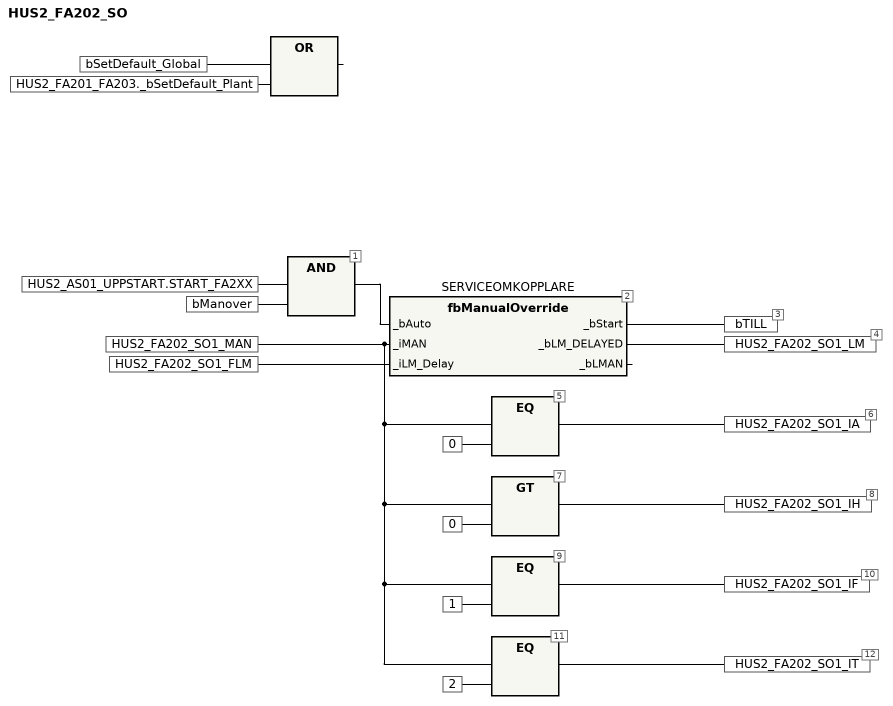
_CFC_ (* Continuous Function Chart, elements in execution order *)
#0 OR(bSetDefault_Global, HUS2_FA201_FA203._bSetDefault_Plant)
#1 AND(HUS2_AS01_UPPSTART.START_FA2XX, bManover)
#2 SERVICEOMKOPPLARE:fbManualOverride(_bAuto: #1, _iMAN: HUS2_FA202_SO1_MAN, _iLM_Delay: HUS2_FA202_SO1_FLM)
#3 bTILL <= #2._bStart
#4 HUS2_FA202_SO1_LM <= #2._bLM_DELAYED
#5 EQ(HUS2_FA202_SO1_MAN, 0)
#6 HUS2_FA202_SO1_IA <= #5
#7 GT(HUS2_FA202_SO1_MAN, 0)
#8 HUS2_FA202_SO1_IH <= #7
#9 EQ(HUS2_FA202_SO1_MAN, 1)
#10 HUS2_FA202_SO1_IF <= #9
#11 EQ(HUS2_FA202_SO1_MAN, 2)
#12 HUS2_FA202_SO1_IT <= #11
_END_CFC_
(* the same logic as Structured Text *)
(* result unused: bSetDefault_Global OR HUS2_FA201_FA203._bSetDefault_Plant *)
SERVICEOMKOPPLARE(_bAuto := HUS2_AS01_UPPSTART.START_FA2XX AND bManover, _iMAN := HUS2_FA202_SO1_MAN, _iLM_Delay := HUS2_FA202_SO1_FLM);
bTILL := SERVICEOMKOPPLARE._bStart;
HUS2_FA202_SO1_LM := SERVICEOMKOPPLARE._bLM_DELAYED;
HUS2_FA202_SO1_IA := HUS2_FA202_SO1_MAN = 0;
HUS2_FA202_SO1_IH := HUS2_FA202_SO1_MAN > 0;
HUS2_FA202_SO1_IF := HUS2_FA202_SO1_MAN = 1;
HUS2_FA202_SO1_IT := HUS2_FA202_SO1_MAN = 2;
END_PROGRAM

(* POU SYSTEM/FA201, FA202, FA203/Fläktstyr/HUS2_FA202_FF01, CFC *)
PROGRAM HUS2_FA202_FF01

VAR
	MANHAND: fbManualOverride;





END_VAR
VAR

END_VAR

VAR_INPUT
	_bAuto							:BOOL;(* enable function block *)
END_VAR

VAR_OUTPUT
	_bMANOVER						:BOOL;
	_bLHAND							:BOOL;
END_VAR
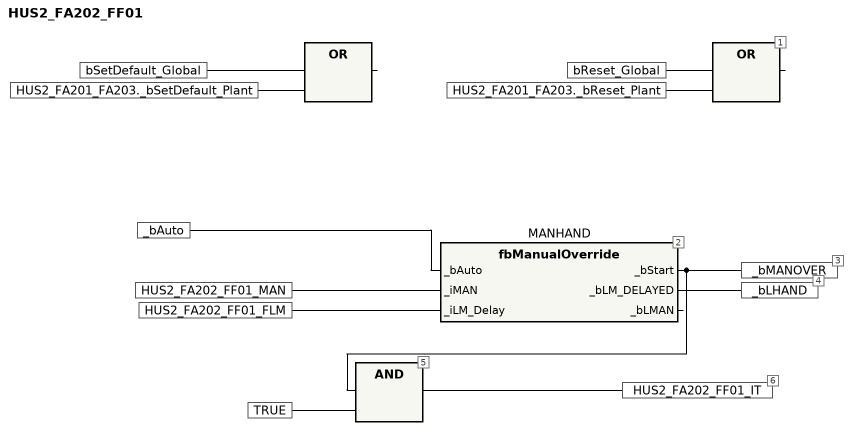
_CFC_ (* Continuous Function Chart, elements in execution order *)
#0 OR(bSetDefault_Global, HUS2_FA201_FA203._bSetDefault_Plant)
#1 OR(bReset_Global, HUS2_FA201_FA203._bReset_Plant)
#2 MANHAND:fbManualOverride(_bAuto: _bAuto, _iMAN: HUS2_FA202_FF01_MAN, _iLM_Delay: HUS2_FA202_FF01_FLM)
#3 _bMANOVER <= #2._bStart
#4 _bLHAND <= #2._bLM_DELAYED
#5 AND(#2._bStart, TRUE)
#6 HUS2_FA202_FF01_IT <= #5
_END_CFC_
(* the same logic as Structured Text *)
(* result unused: bSetDefault_Global OR HUS2_FA201_FA203._bSetDefault_Plant *)
(* result unused: bReset_Global OR HUS2_FA201_FA203._bReset_Plant *)
MANHAND(_bAuto := _bAuto, _iMAN := HUS2_FA202_FF01_MAN, _iLM_Delay := HUS2_FA202_FF01_FLM);
_bMANOVER := MANHAND._bStart;
_bLHAND := MANHAND._bLM_DELAYED;
HUS2_FA202_FF01_IT := MANHAND._bStart AND TRUE;
END_PROGRAM

(* POU SYSTEM/FA201, FA202, FA203/Fläktstyr/HUS2_FA202_FF01_REGLERING, CFC *)
PROGRAM HUS2_FA202_FF01_REGLERING

VAR
	SETRESET: SR;
END_VAR

VAR_INPUT
	bStartFlakt			:BOOL;
	rMV				:REAL;
	rStartForc			:REAL;
	rStoppForc		:REAL;
	rGrundBV			:REAL;
	rForcBV			:REAL;
	bLG				:BOOL;

END_VAR

VAR_OUTPUT
	rSV			:REAL;

END_VAR
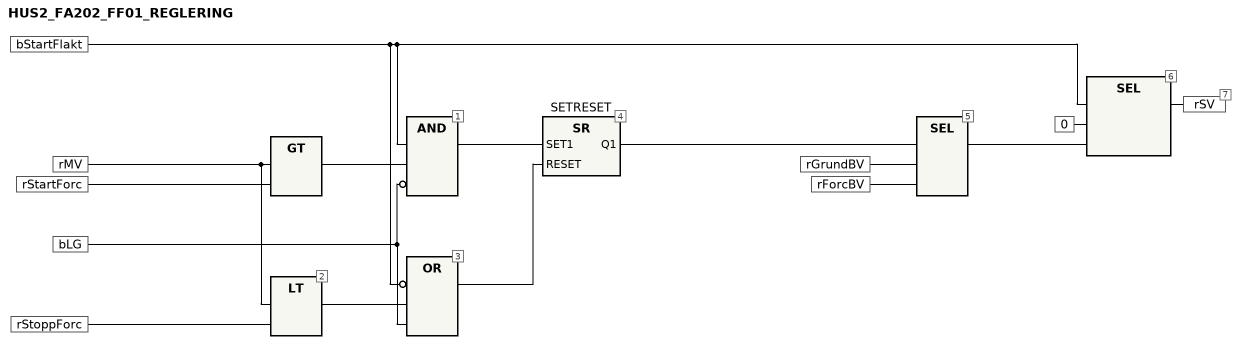
_CFC_ (* Continuous Function Chart, elements in execution order *)
#0 GT(rMV, rStartForc)
#1 AND(bStartFlakt, #0, NOT bLG)
#2 LT(rMV, rStoppForc)
#3 OR(NOT bStartFlakt, #2, bLG)
#4 SETRESET:SR(SET1: #1, RESET: #3)
#5 SEL(#4.Q1, rGrundBV, rForcBV)
#6 SEL(bStartFlakt, 0, #5)
#7 rSV <= #6
_END_CFC_
(* the same logic as Structured Text *)
SETRESET(SET1 := bStartFlakt AND (rMV > rStartForc) AND NOT bLG, RESET := NOT bStartFlakt OR (rMV < rStoppForc) OR bLG);
rSV := SEL(bStartFlakt, 0, SEL(SETRESET.Q1, rGrundBV, rForcBV));
END_PROGRAM

(* POU SYSTEM/FA201, FA202, FA203/Larm/HUS2_FA202_GT51_LARM, FAI *)
PROGRAM HUS2_FA202_GT51_LARM

VAR_OUTPUT
	_bLSumma					: BOOL;	(*Summalarm*)

END_VAR
VAR

	_bSetDefault: 				BOOL;		(*Se default values*)
	fbLarm: fbAvvikelselarm;


	fbHigh: FB_HVACPersistent_Real;
	fbAlarmDelayLH: FB_HVACPersistent_Int;


END_VAR
(* body not read: cfc97 *)
END_PROGRAM

(* POU SYSTEM/FA201, FA202, FA203/HUS2_FA203_SO, CFC *)
PROGRAM HUS2_FA203_SO
VAR_INPUT

	bManover: BOOL;
END_VAR

VAR
	SERVICEOMKOPPLARE: fbManualOverride;

	UPPSTARTSSEKVENSIERING: BOOL;
END_VAR

VAR_OUTPUT
	bTILL:BOOL;

END_VAR
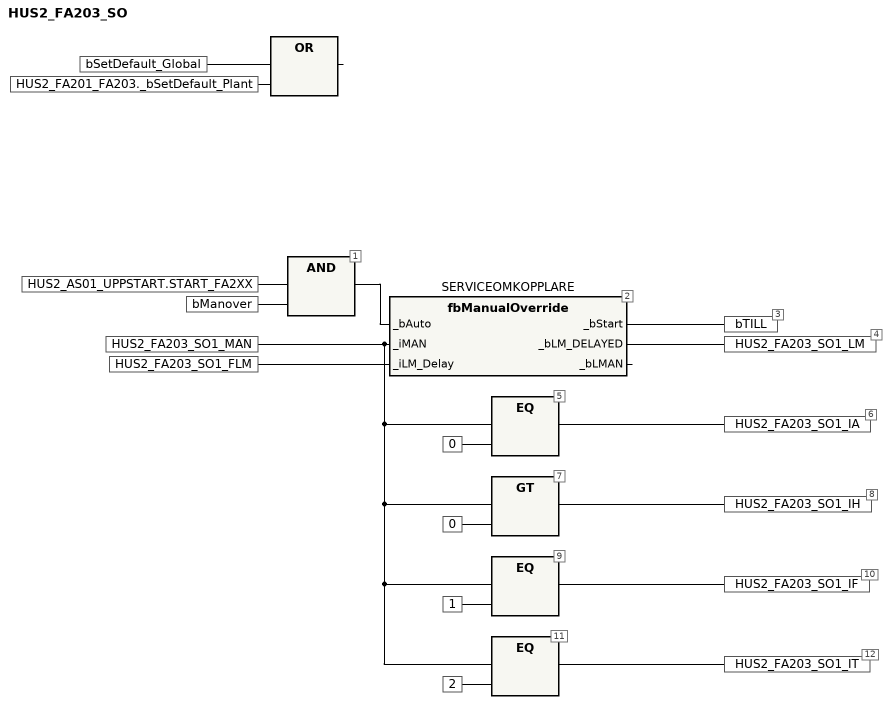
_CFC_ (* Continuous Function Chart, elements in execution order *)
#0 OR(bSetDefault_Global, HUS2_FA201_FA203._bSetDefault_Plant)
#1 AND(HUS2_AS01_UPPSTART.START_FA2XX, bManover)
#2 SERVICEOMKOPPLARE:fbManualOverride(_bAuto: #1, _iMAN: HUS2_FA203_SO1_MAN, _iLM_Delay: HUS2_FA203_SO1_FLM)
#3 bTILL <= #2._bStart
#4 HUS2_FA203_SO1_LM <= #2._bLM_DELAYED
#5 EQ(HUS2_FA203_SO1_MAN, 0)
#6 HUS2_FA203_SO1_IA <= #5
#7 GT(HUS2_FA203_SO1_MAN, 0)
#8 HUS2_FA203_SO1_IH <= #7
#9 EQ(HUS2_FA203_SO1_MAN, 1)
#10 HUS2_FA203_SO1_IF <= #9
#11 EQ(HUS2_FA203_SO1_MAN, 2)
#12 HUS2_FA203_SO1_IT <= #11
_END_CFC_
(* the same logic as Structured Text *)
(* result unused: bSetDefault_Global OR HUS2_FA201_FA203._bSetDefault_Plant *)
SERVICEOMKOPPLARE(_bAuto := HUS2_AS01_UPPSTART.START_FA2XX AND bManover, _iMAN := HUS2_FA203_SO1_MAN, _iLM_Delay := HUS2_FA203_SO1_FLM);
bTILL := SERVICEOMKOPPLARE._bStart;
HUS2_FA203_SO1_LM := SERVICEOMKOPPLARE._bLM_DELAYED;
HUS2_FA203_SO1_IA := HUS2_FA203_SO1_MAN = 0;
HUS2_FA203_SO1_IH := HUS2_FA203_SO1_MAN > 0;
HUS2_FA203_SO1_IF := HUS2_FA203_SO1_MAN = 1;
HUS2_FA203_SO1_IT := HUS2_FA203_SO1_MAN = 2;
END_PROGRAM

(* POU SYSTEM/FA201, FA202, FA203/Fläktstyr/HUS2_FA203_FF01, CFC *)
PROGRAM HUS2_FA203_FF01

VAR
	MANHAND: fbManualOverride;





END_VAR
VAR

END_VAR

VAR_INPUT
	_bAuto							:BOOL;(* enable function block *)
END_VAR

VAR_OUTPUT
	_bMANOVER						:BOOL;
	_bLHAND							:BOOL;
END_VAR
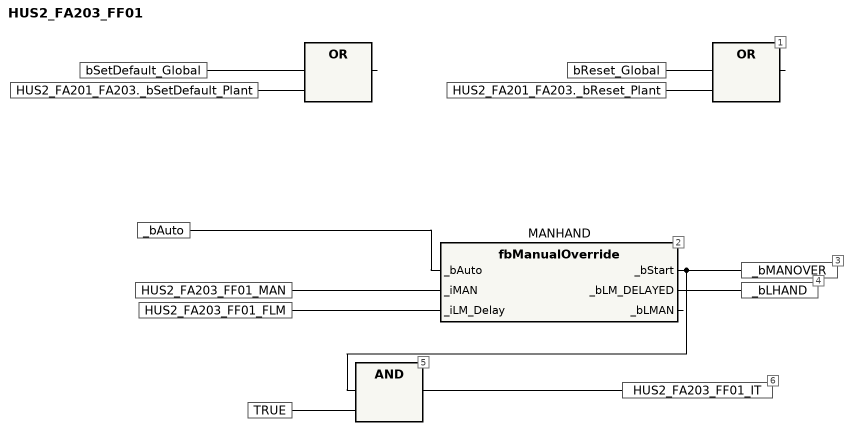
_CFC_ (* Continuous Function Chart, elements in execution order *)
#0 OR(bSetDefault_Global, HUS2_FA201_FA203._bSetDefault_Plant)
#1 OR(bReset_Global, HUS2_FA201_FA203._bReset_Plant)
#2 MANHAND:fbManualOverride(_bAuto: _bAuto, _iMAN: HUS2_FA203_FF01_MAN, _iLM_Delay: HUS2_FA203_FF01_FLM)
#3 _bMANOVER <= #2._bStart
#4 _bLHAND <= #2._bLM_DELAYED
#5 AND(#2._bStart, TRUE)
#6 HUS2_FA203_FF01_IT <= #5
_END_CFC_
(* the same logic as Structured Text *)
(* result unused: bSetDefault_Global OR HUS2_FA201_FA203._bSetDefault_Plant *)
(* result unused: bReset_Global OR HUS2_FA201_FA203._bReset_Plant *)
MANHAND(_bAuto := _bAuto, _iMAN := HUS2_FA203_FF01_MAN, _iLM_Delay := HUS2_FA203_FF01_FLM);
_bMANOVER := MANHAND._bStart;
_bLHAND := MANHAND._bLM_DELAYED;
HUS2_FA203_FF01_IT := MANHAND._bStart AND TRUE;
END_PROGRAM

(* POU SYSTEM/FA201, FA202, FA203/Fläktstyr/HUS2_FA203_FF01_REGLERING, CFC *)
PROGRAM HUS2_FA203_FF01_REGLERING

VAR
	SETRESET: SR;
END_VAR

VAR_INPUT
	bStartFlakt			:BOOL;
	rMV				:REAL;
	rStartForc			:REAL;
	rStoppForc		:REAL;
	rGrundBV			:REAL;
	rForcBV			:REAL;
	bLG				:BOOL;

END_VAR

VAR_OUTPUT
	rSV			:REAL;

END_VAR
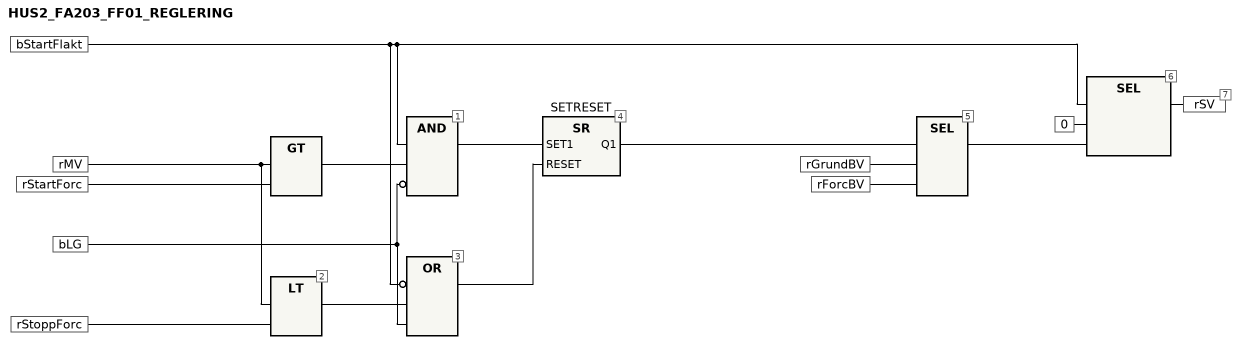
_CFC_ (* Continuous Function Chart, elements in execution order *)
#0 GT(rMV, rStartForc)
#1 AND(bStartFlakt, #0, NOT bLG)
#2 LT(rMV, rStoppForc)
#3 OR(NOT bStartFlakt, #2, bLG)
#4 SETRESET:SR(SET1: #1, RESET: #3)
#5 SEL(#4.Q1, rGrundBV, rForcBV)
#6 SEL(bStartFlakt, 0, #5)
#7 rSV <= #6
_END_CFC_
(* the same logic as Structured Text *)
SETRESET(SET1 := bStartFlakt AND (rMV > rStartForc) AND NOT bLG, RESET := NOT bStartFlakt OR (rMV < rStoppForc) OR bLG);
rSV := SEL(bStartFlakt, 0, SEL(SETRESET.Q1, rGrundBV, rForcBV));
END_PROGRAM

(* POU SYSTEM/FA201, FA202, FA203/Larm/HUS2_FA203_GT51_LARM, FAI *)
PROGRAM HUS2_FA203_GT51_LARM

VAR_OUTPUT
	_bLSumma					: BOOL;	(*Summalarm*)

END_VAR
VAR

	_bSetDefault: 				BOOL;		(*Se default values*)
	fbLarm: fbAvvikelselarm;


	fbHigh: FB_HVACPersistent_Real;
	fbAlarmDelayLH: FB_HVACPersistent_Int;


END_VAR
(* body not read: cfc97 *)
END_PROGRAM

(* POU SYSTEM/FA301, FA302, FA303/HUS3_FA301_FA303, CFC *)
PROGRAM HUS3_FA301_FA303
VAR
	_bSetDefault_Plant		:BOOL;
	_bReset_Plant				:BOOL;

	HUS3_FA301_FF01_M: BOOL;
	HUS3_FA302_FF01_M: BOOL;
	HUS3_FA303_FF01_M: BOOL;
	OVERRIDE_FA301: fbManualOverrideAnalog;
	OVERRIDE_FA302: fbManualOverrideAnalog;
	OVERRIDE_FA303: fbManualOverrideAnalog;
END_VAR
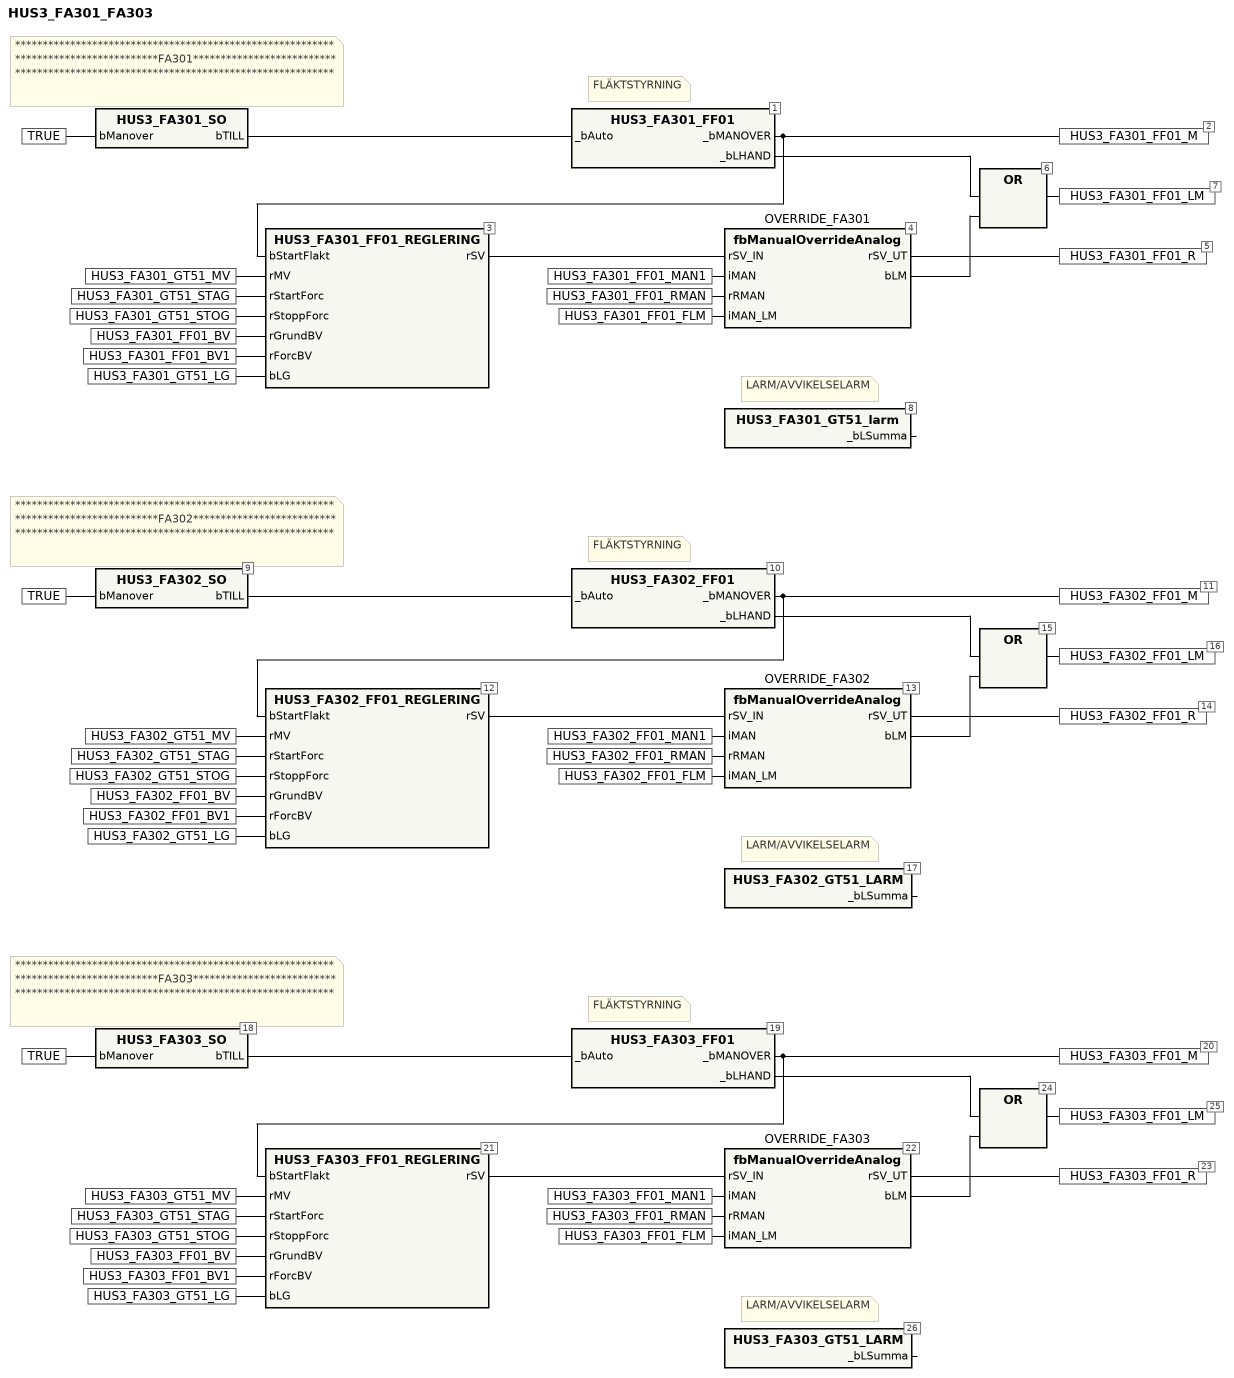
_CFC_ (* Continuous Function Chart, elements in execution order *)
(* LARM/AVVIKELSELARM *)
(* FLÄKTSTYRNING *)
(* ************************************************************************************FA303************************************************************************************ *)
(* LARM/AVVIKELSELARM *)
(* FLÄKTSTYRNING *)
(* LARM/AVVIKELSELARM *)
(* FLÄKTSTYRNING *)
(* ************************************************************************************FA302************************************************************************************ *)
(* ************************************************************************************FA301************************************************************************************ *)
#0 HUS3_FA301_SO(bManover: TRUE)
#1 HUS3_FA301_FF01(_bAuto: #0.bTILL)
#2 HUS3_FA301_FF01_M <= #1._bMANOVER
#3 HUS3_FA301_FF01_REGLERING(bStartFlakt: #1._bMANOVER, rMV: HUS3_FA301_GT51_MV, rStartForc: HUS3_FA301_GT51_STAG, rStoppForc: HUS3_FA301_GT51_STOG, rGrundBV: HUS3_FA301_FF01_BV, rForcBV: HUS3_FA301_FF01_BV1, bLG: HUS3_FA301_GT51_LG)
#4 OVERRIDE_FA301:fbManualOverrideAnalog(rSV_IN: #3.rSV, iMAN: HUS3_FA301_FF01_MAN1, rRMAN: HUS3_FA301_FF01_RMAN, iMAN_LM: HUS3_FA301_FF01_FLM)
#5 HUS3_FA301_FF01_R <= #4.rSV_UT
#6 OR(#1._bLHAND, #4.bLM)
#7 HUS3_FA301_FF01_LM <= #6
#8 HUS3_FA301_GT51_larm()
#9 HUS3_FA302_SO(bManover: TRUE)
#10 HUS3_FA302_FF01(_bAuto: #9.bTILL)
#11 HUS3_FA302_FF01_M <= #10._bMANOVER
#12 HUS3_FA302_FF01_REGLERING(bStartFlakt: #10._bMANOVER, rMV: HUS3_FA302_GT51_MV, rStartForc: HUS3_FA302_GT51_STAG, rStoppForc: HUS3_FA302_GT51_STOG, rGrundBV: HUS3_FA302_FF01_BV, rForcBV: HUS3_FA302_FF01_BV1, bLG: HUS3_FA302_GT51_LG)
#13 OVERRIDE_FA302:fbManualOverrideAnalog(rSV_IN: #12.rSV, iMAN: HUS3_FA302_FF01_MAN1, rRMAN: HUS3_FA302_FF01_RMAN, iMAN_LM: HUS3_FA302_FF01_FLM)
#14 HUS3_FA302_FF01_R <= #13.rSV_UT
#15 OR(#10._bLHAND, #13.bLM)
#16 HUS3_FA302_FF01_LM <= #15
#17 HUS3_FA302_GT51_LARM()
#18 HUS3_FA303_SO(bManover: TRUE)
#19 HUS3_FA303_FF01(_bAuto: #18.bTILL)
#20 HUS3_FA303_FF01_M <= #19._bMANOVER
#21 HUS3_FA303_FF01_REGLERING(bStartFlakt: #19._bMANOVER, rMV: HUS3_FA303_GT51_MV, rStartForc: HUS3_FA303_GT51_STAG, rStoppForc: HUS3_FA303_GT51_STOG, rGrundBV: HUS3_FA303_FF01_BV, rForcBV: HUS3_FA303_FF01_BV1, bLG: HUS3_FA303_GT51_LG)
#22 OVERRIDE_FA303:fbManualOverrideAnalog(rSV_IN: #21.rSV, iMAN: HUS3_FA303_FF01_MAN1, rRMAN: HUS3_FA303_FF01_RMAN, iMAN_LM: HUS3_FA303_FF01_FLM)
#23 HUS3_FA303_FF01_R <= #22.rSV_UT
#24 OR(#19._bLHAND, #22.bLM)
#25 HUS3_FA303_FF01_LM <= #24
#26 HUS3_FA303_GT51_LARM()
_END_CFC_
(* the same logic as Structured Text *)
(* LARM/AVVIKELSELARM *)
(* FLÄKTSTYRNING *)
(* ************************************************************************************FA303************************************************************************************ *)
(* LARM/AVVIKELSELARM *)
(* FLÄKTSTYRNING *)
(* LARM/AVVIKELSELARM *)
(* FLÄKTSTYRNING *)
(* ************************************************************************************FA302************************************************************************************ *)
(* ************************************************************************************FA301************************************************************************************ *)
HUS3_FA301_SO(bManover := TRUE);
HUS3_FA301_FF01(_bAuto := HUS3_FA301_SO.bTILL);
HUS3_FA301_FF01_M := HUS3_FA301_FF01._bMANOVER;
HUS3_FA301_FF01_REGLERING(bStartFlakt := HUS3_FA301_FF01._bMANOVER, rMV := HUS3_FA301_GT51_MV, rStartForc := HUS3_FA301_GT51_STAG, rStoppForc := HUS3_FA301_GT51_STOG, rGrundBV := HUS3_FA301_FF01_BV, rForcBV := HUS3_FA301_FF01_BV1, bLG := HUS3_FA301_GT51_LG);
OVERRIDE_FA301(rSV_IN := HUS3_FA301_FF01_REGLERING.rSV, iMAN := HUS3_FA301_FF01_MAN1, rRMAN := HUS3_FA301_FF01_RMAN, iMAN_LM := HUS3_FA301_FF01_FLM);
HUS3_FA301_FF01_R := OVERRIDE_FA301.rSV_UT;
HUS3_FA301_FF01_LM := HUS3_FA301_FF01._bLHAND OR OVERRIDE_FA301.bLM;
HUS3_FA301_GT51_larm();
HUS3_FA302_SO(bManover := TRUE);
HUS3_FA302_FF01(_bAuto := HUS3_FA302_SO.bTILL);
HUS3_FA302_FF01_M := HUS3_FA302_FF01._bMANOVER;
HUS3_FA302_FF01_REGLERING(bStartFlakt := HUS3_FA302_FF01._bMANOVER, rMV := HUS3_FA302_GT51_MV, rStartForc := HUS3_FA302_GT51_STAG, rStoppForc := HUS3_FA302_GT51_STOG, rGrundBV := HUS3_FA302_FF01_BV, rForcBV := HUS3_FA302_FF01_BV1, bLG := HUS3_FA302_GT51_LG);
OVERRIDE_FA302(rSV_IN := HUS3_FA302_FF01_REGLERING.rSV, iMAN := HUS3_FA302_FF01_MAN1, rRMAN := HUS3_FA302_FF01_RMAN, iMAN_LM := HUS3_FA302_FF01_FLM);
HUS3_FA302_FF01_R := OVERRIDE_FA302.rSV_UT;
HUS3_FA302_FF01_LM := HUS3_FA302_FF01._bLHAND OR OVERRIDE_FA302.bLM;
HUS3_FA302_GT51_LARM();
HUS3_FA303_SO(bManover := TRUE);
HUS3_FA303_FF01(_bAuto := HUS3_FA303_SO.bTILL);
HUS3_FA303_FF01_M := HUS3_FA303_FF01._bMANOVER;
HUS3_FA303_FF01_REGLERING(bStartFlakt := HUS3_FA303_FF01._bMANOVER, rMV := HUS3_FA303_GT51_MV, rStartForc := HUS3_FA303_GT51_STAG, rStoppForc := HUS3_FA303_GT51_STOG, rGrundBV := HUS3_FA303_FF01_BV, rForcBV := HUS3_FA303_FF01_BV1, bLG := HUS3_FA303_GT51_LG);
OVERRIDE_FA303(rSV_IN := HUS3_FA303_FF01_REGLERING.rSV, iMAN := HUS3_FA303_FF01_MAN1, rRMAN := HUS3_FA303_FF01_RMAN, iMAN_LM := HUS3_FA303_FF01_FLM);
HUS3_FA303_FF01_R := OVERRIDE_FA303.rSV_UT;
HUS3_FA303_FF01_LM := HUS3_FA303_FF01._bLHAND OR OVERRIDE_FA303.bLM;
HUS3_FA303_GT51_LARM();
END_PROGRAM

(* POU SYSTEM/FA301, FA302, FA303/HUS3_FA301_SO, CFC *)
PROGRAM HUS3_FA301_SO
VAR_INPUT

	bManover: BOOL;
END_VAR

VAR
	SERVICEOMKOPPLARE: fbManualOverride;

	UPPSTARTSSEKVENSIERING: BOOL;
END_VAR

VAR_OUTPUT
	bTILL:BOOL;

END_VAR
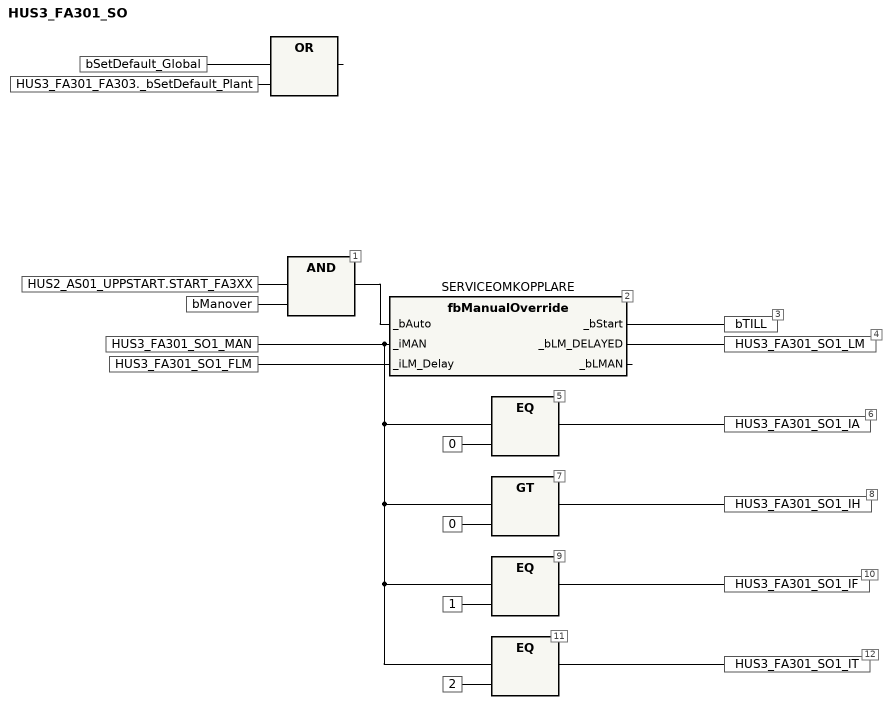
_CFC_ (* Continuous Function Chart, elements in execution order *)
#0 OR(bSetDefault_Global, HUS3_FA301_FA303._bSetDefault_Plant)
#1 AND(HUS2_AS01_UPPSTART.START_FA3XX, bManover)
#2 SERVICEOMKOPPLARE:fbManualOverride(_bAuto: #1, _iMAN: HUS3_FA301_SO1_MAN, _iLM_Delay: HUS3_FA301_SO1_FLM)
#3 bTILL <= #2._bStart
#4 HUS3_FA301_SO1_LM <= #2._bLM_DELAYED
#5 EQ(HUS3_FA301_SO1_MAN, 0)
#6 HUS3_FA301_SO1_IA <= #5
#7 GT(HUS3_FA301_SO1_MAN, 0)
#8 HUS3_FA301_SO1_IH <= #7
#9 EQ(HUS3_FA301_SO1_MAN, 1)
#10 HUS3_FA301_SO1_IF <= #9
#11 EQ(HUS3_FA301_SO1_MAN, 2)
#12 HUS3_FA301_SO1_IT <= #11
_END_CFC_
(* the same logic as Structured Text *)
(* result unused: bSetDefault_Global OR HUS3_FA301_FA303._bSetDefault_Plant *)
SERVICEOMKOPPLARE(_bAuto := HUS2_AS01_UPPSTART.START_FA3XX AND bManover, _iMAN := HUS3_FA301_SO1_MAN, _iLM_Delay := HUS3_FA301_SO1_FLM);
bTILL := SERVICEOMKOPPLARE._bStart;
HUS3_FA301_SO1_LM := SERVICEOMKOPPLARE._bLM_DELAYED;
HUS3_FA301_SO1_IA := HUS3_FA301_SO1_MAN = 0;
HUS3_FA301_SO1_IH := HUS3_FA301_SO1_MAN > 0;
HUS3_FA301_SO1_IF := HUS3_FA301_SO1_MAN = 1;
HUS3_FA301_SO1_IT := HUS3_FA301_SO1_MAN = 2;
END_PROGRAM

(* POU SYSTEM/FA301, FA302, FA303/Fläktstyr/HUS3_FA301_FF01, CFC *)
PROGRAM HUS3_FA301_FF01

VAR
	MANHAND: fbManualOverride;





END_VAR
VAR

END_VAR

VAR_INPUT
	_bAuto							:BOOL;(* enable function block *)
END_VAR

VAR_OUTPUT
	_bMANOVER						:BOOL;
	_bLHAND							:BOOL;
END_VAR
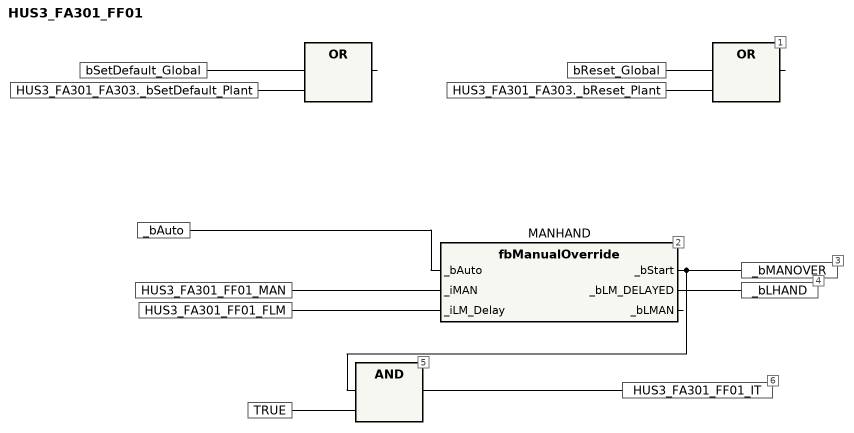
_CFC_ (* Continuous Function Chart, elements in execution order *)
#0 OR(bSetDefault_Global, HUS3_FA301_FA303._bSetDefault_Plant)
#1 OR(bReset_Global, HUS3_FA301_FA303._bReset_Plant)
#2 MANHAND:fbManualOverride(_bAuto: _bAuto, _iMAN: HUS3_FA301_FF01_MAN, _iLM_Delay: HUS3_FA301_FF01_FLM)
#3 _bMANOVER <= #2._bStart
#4 _bLHAND <= #2._bLM_DELAYED
#5 AND(#2._bStart, TRUE)
#6 HUS3_FA301_FF01_IT <= #5
_END_CFC_
(* the same logic as Structured Text *)
(* result unused: bSetDefault_Global OR HUS3_FA301_FA303._bSetDefault_Plant *)
(* result unused: bReset_Global OR HUS3_FA301_FA303._bReset_Plant *)
MANHAND(_bAuto := _bAuto, _iMAN := HUS3_FA301_FF01_MAN, _iLM_Delay := HUS3_FA301_FF01_FLM);
_bMANOVER := MANHAND._bStart;
_bLHAND := MANHAND._bLM_DELAYED;
HUS3_FA301_FF01_IT := MANHAND._bStart AND TRUE;
END_PROGRAM

(* POU SYSTEM/FA301, FA302, FA303/Fläktstyr/HUS3_FA301_FF01_REGLERING, CFC *)
PROGRAM HUS3_FA301_FF01_REGLERING

VAR
	SETRESET: SR;
END_VAR

VAR_INPUT
	bStartFlakt			:BOOL;
	rMV				:REAL;
	rStartForc			:REAL;
	rStoppForc		:REAL;
	rGrundBV			:REAL;
	rForcBV			:REAL;
	bLG				:BOOL;

END_VAR

VAR_OUTPUT
	rSV			:REAL;

END_VAR
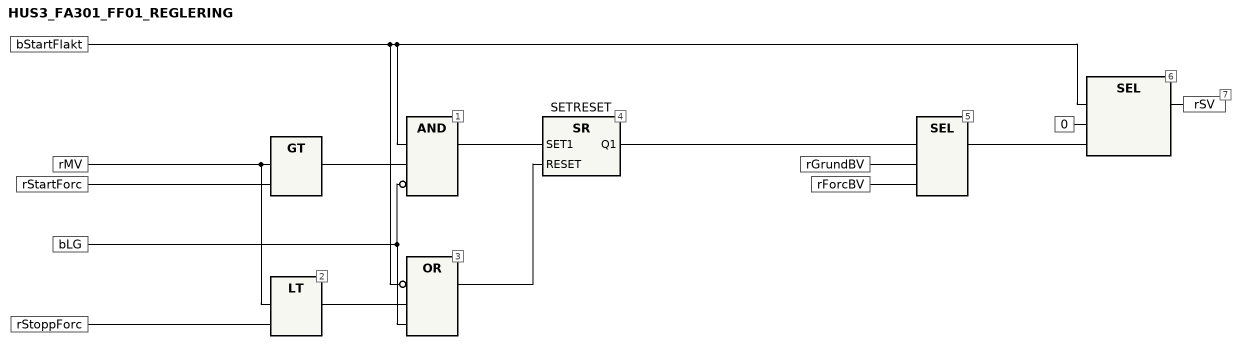
_CFC_ (* Continuous Function Chart, elements in execution order *)
#0 GT(rMV, rStartForc)
#1 AND(bStartFlakt, #0, NOT bLG)
#2 LT(rMV, rStoppForc)
#3 OR(NOT bStartFlakt, #2, bLG)
#4 SETRESET:SR(SET1: #1, RESET: #3)
#5 SEL(#4.Q1, rGrundBV, rForcBV)
#6 SEL(bStartFlakt, 0, #5)
#7 rSV <= #6
_END_CFC_
(* the same logic as Structured Text *)
SETRESET(SET1 := bStartFlakt AND (rMV > rStartForc) AND NOT bLG, RESET := NOT bStartFlakt OR (rMV < rStoppForc) OR bLG);
rSV := SEL(bStartFlakt, 0, SEL(SETRESET.Q1, rGrundBV, rForcBV));
END_PROGRAM

(* POU SYSTEM/FA301, FA302, FA303/Larm/HUS3_FA301_GT51_LARM, FAI *)
PROGRAM HUS3_FA301_GT51_LARM

VAR_OUTPUT
	_bLSumma					: BOOL;	(*Summalarm*)

END_VAR
VAR

	_bSetDefault: 				BOOL;		(*Se default values*)
	fbLarm: fbAvvikelselarm;


	fbHigh: FB_HVACPersistent_Real;
	fbAlarmDelayLH: FB_HVACPersistent_Int;


END_VAR
(* body not read: cfc97 *)
END_PROGRAM

(* POU SYSTEM/FA301, FA302, FA303/HUS3_FA302_SO, CFC *)
PROGRAM HUS3_FA302_SO
VAR_INPUT

	bManover: BOOL;
END_VAR

VAR
	SERVICEOMKOPPLARE: fbManualOverride;

	UPPSTARTSSEKVENSIERING: BOOL;
END_VAR

VAR_OUTPUT
	bTILL:BOOL;

END_VAR
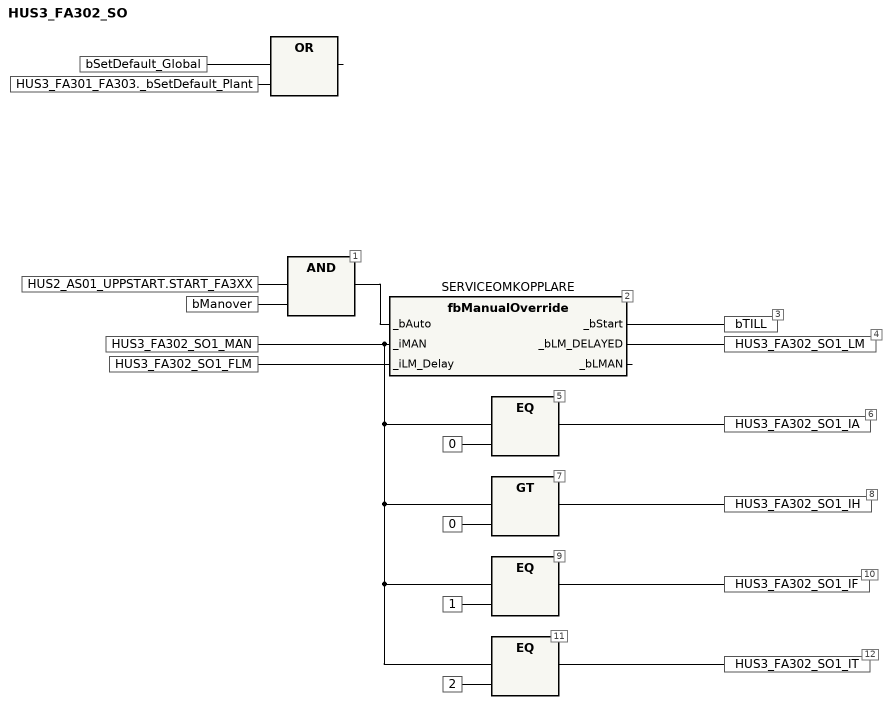
_CFC_ (* Continuous Function Chart, elements in execution order *)
#0 OR(bSetDefault_Global, HUS3_FA301_FA303._bSetDefault_Plant)
#1 AND(HUS2_AS01_UPPSTART.START_FA3XX, bManover)
#2 SERVICEOMKOPPLARE:fbManualOverride(_bAuto: #1, _iMAN: HUS3_FA302_SO1_MAN, _iLM_Delay: HUS3_FA302_SO1_FLM)
#3 bTILL <= #2._bStart
#4 HUS3_FA302_SO1_LM <= #2._bLM_DELAYED
#5 EQ(HUS3_FA302_SO1_MAN, 0)
#6 HUS3_FA302_SO1_IA <= #5
#7 GT(HUS3_FA302_SO1_MAN, 0)
#8 HUS3_FA302_SO1_IH <= #7
#9 EQ(HUS3_FA302_SO1_MAN, 1)
#10 HUS3_FA302_SO1_IF <= #9
#11 EQ(HUS3_FA302_SO1_MAN, 2)
#12 HUS3_FA302_SO1_IT <= #11
_END_CFC_
(* the same logic as Structured Text *)
(* result unused: bSetDefault_Global OR HUS3_FA301_FA303._bSetDefault_Plant *)
SERVICEOMKOPPLARE(_bAuto := HUS2_AS01_UPPSTART.START_FA3XX AND bManover, _iMAN := HUS3_FA302_SO1_MAN, _iLM_Delay := HUS3_FA302_SO1_FLM);
bTILL := SERVICEOMKOPPLARE._bStart;
HUS3_FA302_SO1_LM := SERVICEOMKOPPLARE._bLM_DELAYED;
HUS3_FA302_SO1_IA := HUS3_FA302_SO1_MAN = 0;
HUS3_FA302_SO1_IH := HUS3_FA302_SO1_MAN > 0;
HUS3_FA302_SO1_IF := HUS3_FA302_SO1_MAN = 1;
HUS3_FA302_SO1_IT := HUS3_FA302_SO1_MAN = 2;
END_PROGRAM

(* POU SYSTEM/FA301, FA302, FA303/Fläktstyr/HUS3_FA302_FF01, CFC *)
PROGRAM HUS3_FA302_FF01

VAR
	MANHAND: fbManualOverride;





END_VAR
VAR

END_VAR

VAR_INPUT
	_bAuto							:BOOL;(* enable function block *)
END_VAR

VAR_OUTPUT
	_bMANOVER						:BOOL;
	_bLHAND							:BOOL;
END_VAR
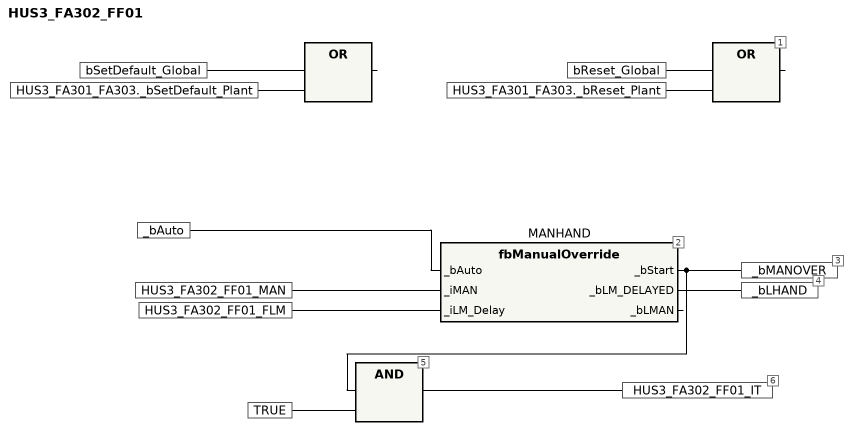
_CFC_ (* Continuous Function Chart, elements in execution order *)
#0 OR(bSetDefault_Global, HUS3_FA301_FA303._bSetDefault_Plant)
#1 OR(bReset_Global, HUS3_FA301_FA303._bReset_Plant)
#2 MANHAND:fbManualOverride(_bAuto: _bAuto, _iMAN: HUS3_FA302_FF01_MAN, _iLM_Delay: HUS3_FA302_FF01_FLM)
#3 _bMANOVER <= #2._bStart
#4 _bLHAND <= #2._bLM_DELAYED
#5 AND(#2._bStart, TRUE)
#6 HUS3_FA302_FF01_IT <= #5
_END_CFC_
(* the same logic as Structured Text *)
(* result unused: bSetDefault_Global OR HUS3_FA301_FA303._bSetDefault_Plant *)
(* result unused: bReset_Global OR HUS3_FA301_FA303._bReset_Plant *)
MANHAND(_bAuto := _bAuto, _iMAN := HUS3_FA302_FF01_MAN, _iLM_Delay := HUS3_FA302_FF01_FLM);
_bMANOVER := MANHAND._bStart;
_bLHAND := MANHAND._bLM_DELAYED;
HUS3_FA302_FF01_IT := MANHAND._bStart AND TRUE;
END_PROGRAM

(* POU SYSTEM/FA301, FA302, FA303/Fläktstyr/HUS3_FA302_FF01_REGLERING, CFC *)
PROGRAM HUS3_FA302_FF01_REGLERING

VAR
	SETRESET: SR;
END_VAR

VAR_INPUT
	bStartFlakt			:BOOL;
	rMV				:REAL;
	rStartForc			:REAL;
	rStoppForc		:REAL;
	rGrundBV			:REAL;
	rForcBV			:REAL;
	bLG				:BOOL;

END_VAR

VAR_OUTPUT
	rSV			:REAL;

END_VAR
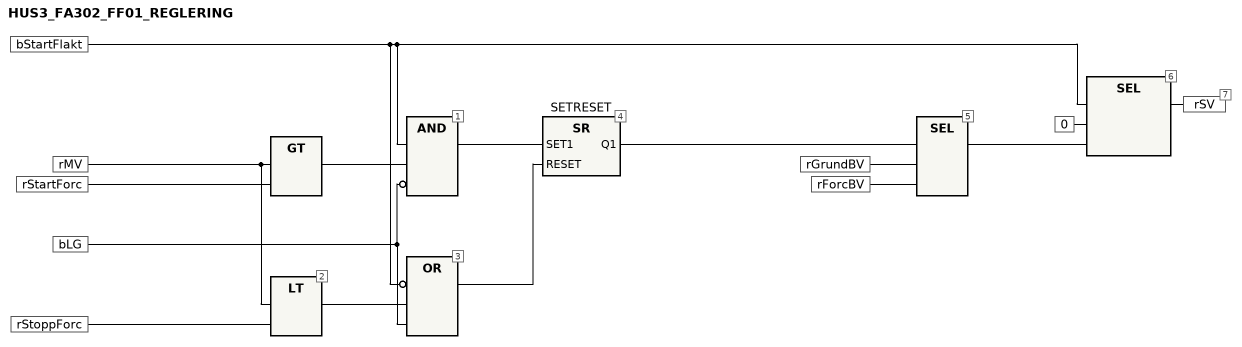
_CFC_ (* Continuous Function Chart, elements in execution order *)
#0 GT(rMV, rStartForc)
#1 AND(bStartFlakt, #0, NOT bLG)
#2 LT(rMV, rStoppForc)
#3 OR(NOT bStartFlakt, #2, bLG)
#4 SETRESET:SR(SET1: #1, RESET: #3)
#5 SEL(#4.Q1, rGrundBV, rForcBV)
#6 SEL(bStartFlakt, 0, #5)
#7 rSV <= #6
_END_CFC_
(* the same logic as Structured Text *)
SETRESET(SET1 := bStartFlakt AND (rMV > rStartForc) AND NOT bLG, RESET := NOT bStartFlakt OR (rMV < rStoppForc) OR bLG);
rSV := SEL(bStartFlakt, 0, SEL(SETRESET.Q1, rGrundBV, rForcBV));
END_PROGRAM

(* POU SYSTEM/FA301, FA302, FA303/Larm/HUS3_FA302_GT51_LARM, FAI *)
PROGRAM HUS3_FA302_GT51_LARM

VAR_OUTPUT
	_bLSumma					: BOOL;	(*Summalarm*)

END_VAR
VAR

	_bSetDefault: 				BOOL;		(*Se default values*)
	fbLarm: fbAvvikelselarm;


	fbHigh: FB_HVACPersistent_Real;
	fbAlarmDelayLH: FB_HVACPersistent_Int;


END_VAR
(* body not read: cfc97 *)
END_PROGRAM

(* POU SYSTEM/FA301, FA302, FA303/HUS3_FA303_SO, CFC *)
PROGRAM HUS3_FA303_SO
VAR_INPUT

	bManover: BOOL;
END_VAR

VAR
	SERVICEOMKOPPLARE: fbManualOverride;

	UPPSTARTSSEKVENSIERING: BOOL;
END_VAR

VAR_OUTPUT
	bTILL:BOOL;

END_VAR
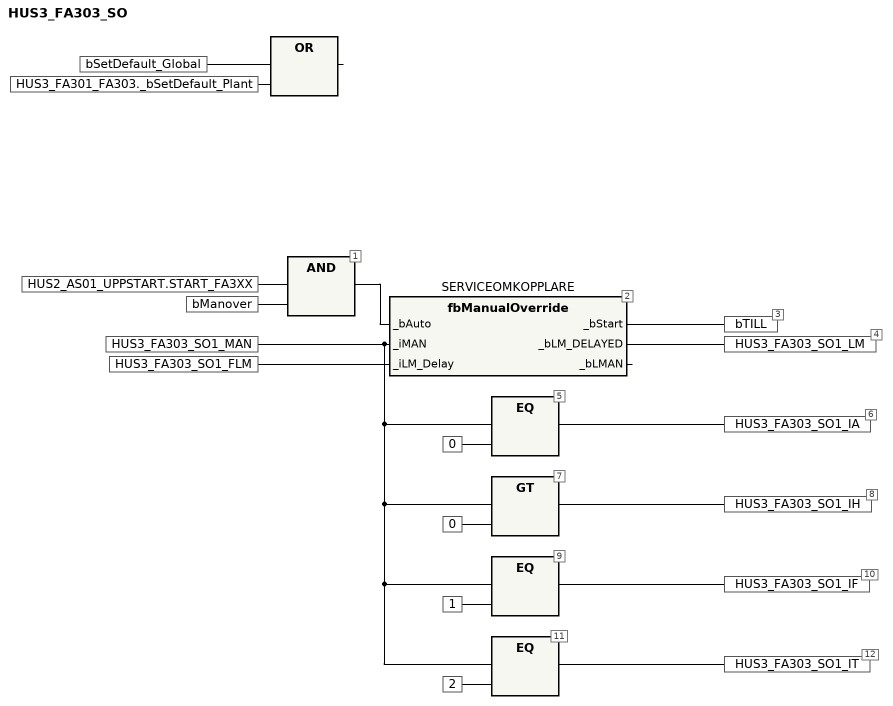
_CFC_ (* Continuous Function Chart, elements in execution order *)
#0 OR(bSetDefault_Global, HUS3_FA301_FA303._bSetDefault_Plant)
#1 AND(HUS2_AS01_UPPSTART.START_FA3XX, bManover)
#2 SERVICEOMKOPPLARE:fbManualOverride(_bAuto: #1, _iMAN: HUS3_FA303_SO1_MAN, _iLM_Delay: HUS3_FA303_SO1_FLM)
#3 bTILL <= #2._bStart
#4 HUS3_FA303_SO1_LM <= #2._bLM_DELAYED
#5 EQ(HUS3_FA303_SO1_MAN, 0)
#6 HUS3_FA303_SO1_IA <= #5
#7 GT(HUS3_FA303_SO1_MAN, 0)
#8 HUS3_FA303_SO1_IH <= #7
#9 EQ(HUS3_FA303_SO1_MAN, 1)
#10 HUS3_FA303_SO1_IF <= #9
#11 EQ(HUS3_FA303_SO1_MAN, 2)
#12 HUS3_FA303_SO1_IT <= #11
_END_CFC_
(* the same logic as Structured Text *)
(* result unused: bSetDefault_Global OR HUS3_FA301_FA303._bSetDefault_Plant *)
SERVICEOMKOPPLARE(_bAuto := HUS2_AS01_UPPSTART.START_FA3XX AND bManover, _iMAN := HUS3_FA303_SO1_MAN, _iLM_Delay := HUS3_FA303_SO1_FLM);
bTILL := SERVICEOMKOPPLARE._bStart;
HUS3_FA303_SO1_LM := SERVICEOMKOPPLARE._bLM_DELAYED;
HUS3_FA303_SO1_IA := HUS3_FA303_SO1_MAN = 0;
HUS3_FA303_SO1_IH := HUS3_FA303_SO1_MAN > 0;
HUS3_FA303_SO1_IF := HUS3_FA303_SO1_MAN = 1;
HUS3_FA303_SO1_IT := HUS3_FA303_SO1_MAN = 2;
END_PROGRAM

(* POU SYSTEM/FA301, FA302, FA303/Fläktstyr/HUS3_FA303_FF01, CFC *)
PROGRAM HUS3_FA303_FF01

VAR
	MANHAND: fbManualOverride;





END_VAR
VAR

END_VAR

VAR_INPUT
	_bAuto							:BOOL;(* enable function block *)
END_VAR

VAR_OUTPUT
	_bMANOVER						:BOOL;
	_bLHAND							:BOOL;
END_VAR
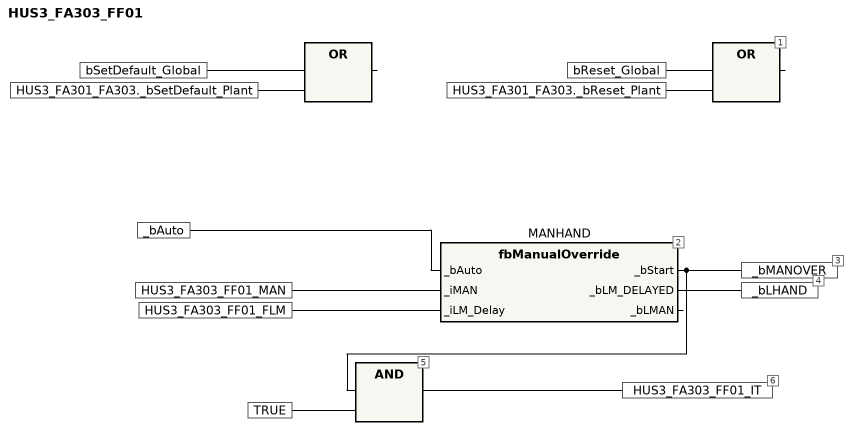
_CFC_ (* Continuous Function Chart, elements in execution order *)
#0 OR(bSetDefault_Global, HUS3_FA301_FA303._bSetDefault_Plant)
#1 OR(bReset_Global, HUS3_FA301_FA303._bReset_Plant)
#2 MANHAND:fbManualOverride(_bAuto: _bAuto, _iMAN: HUS3_FA303_FF01_MAN, _iLM_Delay: HUS3_FA303_FF01_FLM)
#3 _bMANOVER <= #2._bStart
#4 _bLHAND <= #2._bLM_DELAYED
#5 AND(#2._bStart, TRUE)
#6 HUS3_FA303_FF01_IT <= #5
_END_CFC_
(* the same logic as Structured Text *)
(* result unused: bSetDefault_Global OR HUS3_FA301_FA303._bSetDefault_Plant *)
(* result unused: bReset_Global OR HUS3_FA301_FA303._bReset_Plant *)
MANHAND(_bAuto := _bAuto, _iMAN := HUS3_FA303_FF01_MAN, _iLM_Delay := HUS3_FA303_FF01_FLM);
_bMANOVER := MANHAND._bStart;
_bLHAND := MANHAND._bLM_DELAYED;
HUS3_FA303_FF01_IT := MANHAND._bStart AND TRUE;
END_PROGRAM

(* POU SYSTEM/FA301, FA302, FA303/Fläktstyr/HUS3_FA303_FF01_REGLERING, CFC *)
PROGRAM HUS3_FA303_FF01_REGLERING

VAR
	SETRESET: SR;
END_VAR

VAR_INPUT
	bStartFlakt			:BOOL;
	rMV				:REAL;
	rStartForc			:REAL;
	rStoppForc		:REAL;
	rGrundBV			:REAL;
	rForcBV			:REAL;
	bLG				:BOOL;

END_VAR

VAR_OUTPUT
	rSV			:REAL;

END_VAR
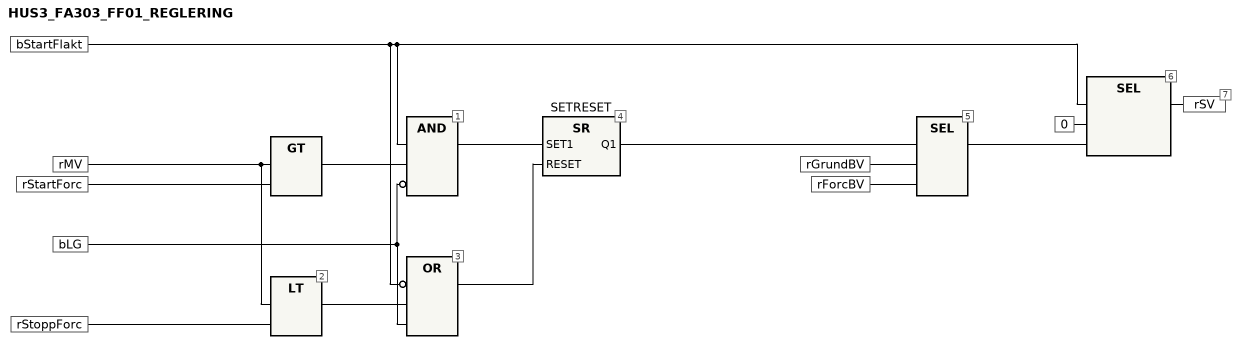
_CFC_ (* Continuous Function Chart, elements in execution order *)
#0 GT(rMV, rStartForc)
#1 AND(bStartFlakt, #0, NOT bLG)
#2 LT(rMV, rStoppForc)
#3 OR(NOT bStartFlakt, #2, bLG)
#4 SETRESET:SR(SET1: #1, RESET: #3)
#5 SEL(#4.Q1, rGrundBV, rForcBV)
#6 SEL(bStartFlakt, 0, #5)
#7 rSV <= #6
_END_CFC_
(* the same logic as Structured Text *)
SETRESET(SET1 := bStartFlakt AND (rMV > rStartForc) AND NOT bLG, RESET := NOT bStartFlakt OR (rMV < rStoppForc) OR bLG);
rSV := SEL(bStartFlakt, 0, SEL(SETRESET.Q1, rGrundBV, rForcBV));
END_PROGRAM

(* POU SYSTEM/FA301, FA302, FA303/Larm/HUS3_FA303_GT51_LARM, FAI *)
PROGRAM HUS3_FA303_GT51_LARM

VAR_OUTPUT
	_bLSumma					: BOOL;	(*Summalarm*)

END_VAR
VAR

	_bSetDefault: 				BOOL;		(*Se default values*)
	fbLarm: fbAvvikelselarm;


	fbHigh: FB_HVACPersistent_Real;
	fbAlarmDelayLH: FB_HVACPersistent_Int;


END_VAR
(* body not read: cfc97 *)
END_PROGRAM

(* POU ReadMe, ST *)
PROGRAM ReadMe
VAR
END_VAR
(*


Oskar Lindström, Automationsbolaget Sverige AB
2020-03-04


*)
END_PROGRAM

(* POU xEgna Funktionsblock/Modbus/Modbusfunktioner_med_Master/_ModbusTCP_Controller, ST *)
FUNCTION_BLOCK _ModbusTCP_Controller

VAR
	stController			: ST_TCP_CONTROLLER:=(iWorkingUnitId:=1);
	pController			: POINTER TO ST_TCP_CONTROLLER;

END_VAR
(* DO NOT CHANGE ANYTHING IN THIS CODE *)

(* Output the pointer to this controller*)
pController := ADR(stController);

(* Do any units exist? *)
IF stController.iNoUnits>0 THEN
	(* Is the current unit done? *)
	IF stController.bUnitIsDone  THEN
		(* Yes, reset the done flag and increase the unit ID counter *)
		stController.bUnitIsDone:=FALSE;
		stController.iWorkingUnitId:=stController.iWorkingUnitId+1;
		(*Handle rollover of the unit ID counter *)
		IF stController.iWorkingUnitId>stController.iNoUnits THEN
			stController.iWorkingUnitId:=1;
		END_IF
	END_IF
END_IF
END_FUNCTION_BLOCK

(* POU xEgna Funktionsblock/Time_to_SCADA/FB_CitectTimeTo_HVAC_1_DATE, ST *)
(*
Funktionsblock för att hantera en tid från Citect/Webport till Beckhoffs tidkanaler
Av: Beckhoff Automation AB Roger Grönvall
Lib: TCHVAC.LIB
*)
FUNCTION_BLOCK FB_CitectTimeTo_HVAC_1_DATE

VAR_INPUT
END_VAR

VAR_IN_OUT
	_iCitect_OnTime:		INT;		(*Time On from HMI*)
	_iCitect_OffTime:		INT;		(*Time Off from HMI*)
END_VAR
VAR_OUTPUT
	_uiOnTime_hh:		UINT;	(*Hours for on time*)
	_uiOnTime_mm:		UINT;	(*Minutes for on time*)
	_uiOffTime_hh:		UINT;	(*Hours for off time*)
	_uiOffTime_mm:		UINT;	(*Minutes for off time*)
	_bEnableTimeCh:		BOOL;	(*Enable timechannel*)
END_VAR
VAR
	iNowOn:				INT;		(*Temp var for on time*)
	iNowOff:				INT;		(*Temp var for off time*)
	fbSaveOnTime:		FB_HVACPersistent_Int;
	fbSaveOffTime:		FB_HVACPersistent_Int;
END_VAR

(*
	This FB converts hmi time from Citect to HVAC TimeChannel
	the input time is an integer. i.e Time 15:46 = _iCitect_OnTime 1546. Then
	the our and minute is extracted to the HVAC time. 
	No erreor handling if time is not in the appropriate range.
	Maybe the persistent data handling for the TC needs to be disabled
*)
(*Get the on time*)
iNowOn := _iCitect_OnTime;
(*Get hour*)
_uiOnTime_hh := iNowOn / 100;
(*Get minute*)
_uiOnTime_mm := iNowOn - ( _uiOnTime_hh * 100);


(*Get the off time*)
iNowOff := _iCitect_OffTime;
(*Get hour*)
_uiOffTime_hh := iNowOff / 100;
(*Get minute*)
_uiOffTime_mm := iNowOff - ( _uiOffTime_hh * 100);


(*Find out if we have some time set, then enable the output*)
IF  _iCitect_OnTime > 0 THEN
	_bEnableTimeCh := TRUE;
ELSE
	_bEnableTimeCh := FALSE;
END_IF


(*Save the on/off time data persistent*)
fbSaveOnTime(bSetDefault:= , iVar_Default:= , iVar:= _iCitect_OnTime );
fbSaveOffTime(bSetDefault:= , iVar_Default:= , iVar:= _iCitect_OffTime );
END_FUNCTION_BLOCK

(* POU xEgna Funktionsblock/fbActiveLG, CFC *)
FUNCTION_BLOCK fbActiveLG
VAR_INPUT
	rMV:REAL;
	rHighLimit:REAL;
	rLowLimit:REAL;
	iLG_FL:INT;
END_VAR
VAR_OUTPUT
	bLG:BOOL;
END_VAR
VAR
	FBTON1: TON;
END_VAR
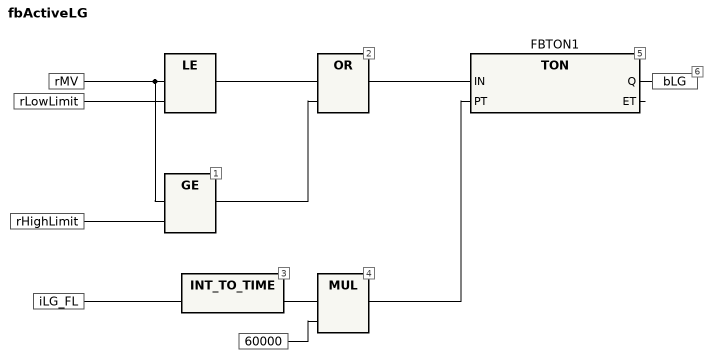
_CFC_ (* Continuous Function Chart, elements in execution order *)
#0 LE(rMV, rLowLimit)
#1 GE(rMV, rHighLimit)
#2 OR(#0, #1)
#3 INT_TO_TIME(iLG_FL)
#4 MUL(#3, 60000)
#5 FBTON1:TON(IN: #2, PT: #4)
#6 bLG <= #5.Q
_END_CFC_
(* the same logic as Structured Text *)
FBTON1(IN := (rMV <= rLowLimit) OR (rMV >= rHighLimit), PT := INT_TO_TIME(iLG_FL) * 60000);
bLG := FBTON1.Q;
END_FUNCTION_BLOCK

(* POU xEgna Funktionsblock/fbAvvikelselarm_SEC, CFC *)
FUNCTION_BLOCK fbAvvikelselarm_SEC
VAR
	TON1: TON;
	TON2: TON;
END_VAR
VAR_INPUT
	_rBB: REAL;
	_rMV: REAL;
	_rLL: REAL;
	_iFLL: INT;
	_rLH: REAL;
	_iFLH: INT;
	_bAktiveraLarm: BOOL;

END_VAR


VAR_OUTPUT
	_bLL: BOOL;
	_bLH: BOOL;
	_bLSummA: BOOL;
END_VAR
VAR (* helpers for the ST form of the networks *)
	_t54 : TIME;
END_VAR
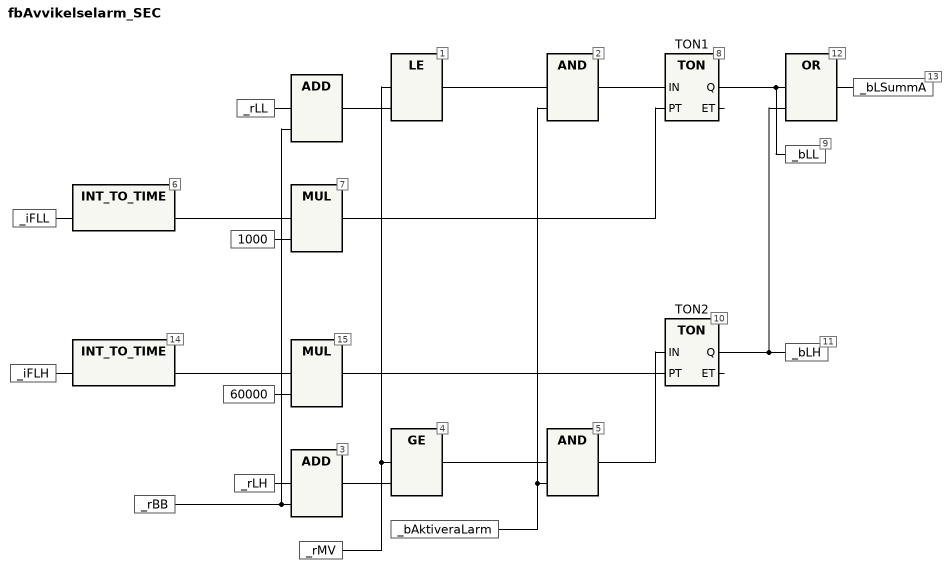
_CFC_ (* Continuous Function Chart, elements in execution order *)
#0 ADD(_rLL, _rBB)
#1 LE(_rMV, #0)
#2 AND(#1, _bAktiveraLarm)
#3 ADD(_rLH, _rBB)
#4 GE(_rMV, #3)
#5 AND(#4, _bAktiveraLarm)
#6 INT_TO_TIME(_iFLL)
#7 MUL(#6, 1000)
#8 TON1:TON(IN: #2, PT: #7)
#9 _bLL <= #8.Q
#10 TON2:TON(IN: #5, PT: #15)
#11 _bLH <= #10.Q
#12 OR(#8.Q, #10.Q)
#13 _bLSummA <= #12
#14 INT_TO_TIME(_iFLH)
#15 MUL(#14, 60000)
_END_CFC_
(* the same logic as Structured Text *)
TON1(IN := (_rMV <= (_rLL + _rBB)) AND _bAktiveraLarm, PT := INT_TO_TIME(_iFLL) * 1000);
_bLL := TON1.Q;
TON2(IN := (_rMV >= (_rLH + _rBB)) AND _bAktiveraLarm, PT := _t54);
_bLH := TON2.Q;
_bLSummA := TON1.Q OR TON2.Q;
_t54 := INT_TO_TIME(_iFLH) * 60000;
END_FUNCTION_BLOCK

(* POU xEgna Funktionsblock/fbAvvikelselarmLA, CFC *)
FUNCTION_BLOCK fbAvvikelselarmLA
VAR
	TON1: TON;
	TON2: TON;
END_VAR
VAR_INPUT
	_rBB: REAL;
	_rMV: REAL;
	_rLA: REAL;
	_iFLA: INT;
	_bAktiveraLarm: BOOL;

END_VAR


VAR_OUTPUT
	_bLA: BOOL;
END_VAR
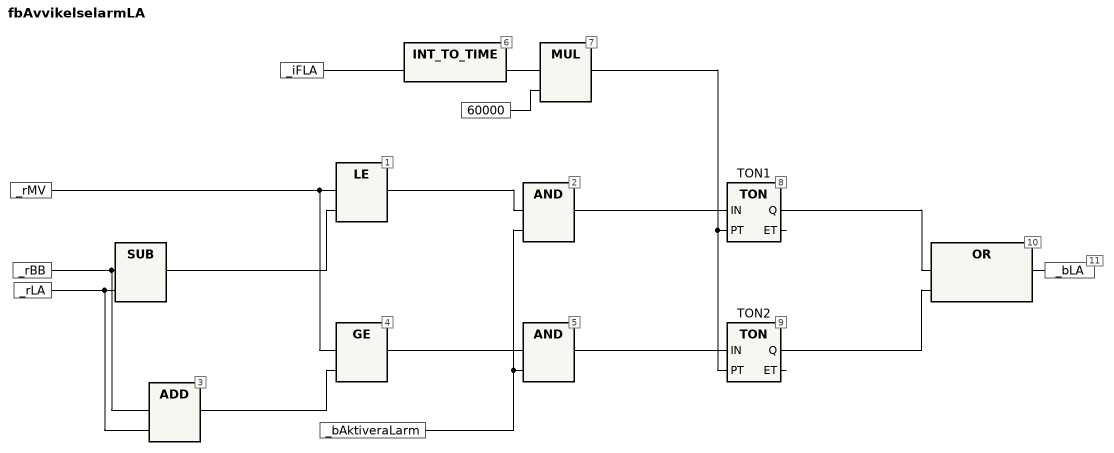
_CFC_ (* Continuous Function Chart, elements in execution order *)
#0 SUB(_rBB, _rLA)
#1 LE(_rMV, #0)
#2 AND(#1, _bAktiveraLarm)
#3 ADD(_rBB, _rLA)
#4 GE(_rMV, #3)
#5 AND(#4, _bAktiveraLarm)
#6 INT_TO_TIME(_iFLA)
#7 MUL(#6, 60000)
#8 TON1:TON(IN: #2, PT: #7)
#9 TON2:TON(IN: #5, PT: #7)
#10 OR(#8.Q, #9.Q)
#11 _bLA <= #10
_END_CFC_
(* the same logic as Structured Text *)
TON1(IN := (_rMV <= (_rBB - _rLA)) AND _bAktiveraLarm, PT := INT_TO_TIME(_iFLA) * 60000);
TON2(IN := (_rMV >= (_rBB + _rLA)) AND _bAktiveraLarm, PT := INT_TO_TIME(_iFLA) * 60000);
_bLA := TON1.Q OR TON2.Q;
END_FUNCTION_BLOCK

(* POU xEgna Funktionsblock/fbINT_TO_SEC, CFC *)
FUNCTION_BLOCK fbINT_TO_SEC
VAR_INPUT
	iSeconds :INT;
END_VAR
VAR_OUTPUT
	tSEC: TIME;
END_VAR
VAR

END_VAR
VAR (* helpers for the ST form of the networks *)
	_t5 : TIME;
END_VAR
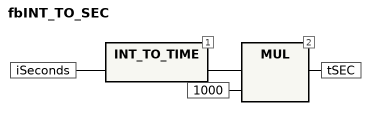
_CFC_ (* Continuous Function Chart, elements in execution order *)
#0 tSEC <= #2
#1 INT_TO_TIME(iSeconds)
#2 MUL(#1, 1000)
_END_CFC_
(* the same logic as Structured Text *)
tSEC := _t5;
_t5 := INT_TO_TIME(iSeconds) * 1000;
END_FUNCTION_BLOCK

(* POU xEgna Funktionsblock/fbMedelBer, CFC *)
FUNCTION_BLOCK fbMedelBer
VAR_INPUT
	_MV1:REAL;
	_MV2:REAL;
	_MV1_L:BOOL;
	_MV2_L:BOOL;
END_VAR
VAR_OUTPUT
	_MV_Medel:REAL;
END_VAR
VAR
END_VAR
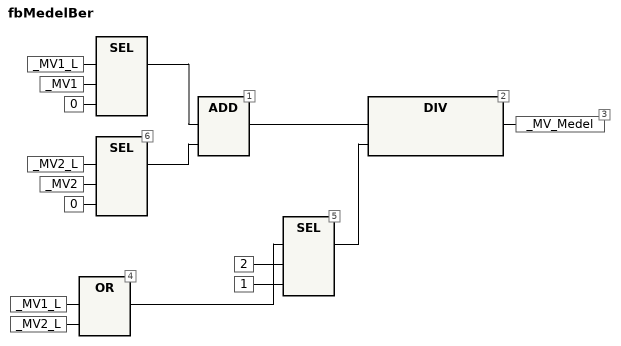
_CFC_ (* Continuous Function Chart, elements in execution order *)
#0 SEL(_MV1_L, _MV1, 0)
#1 ADD(#0, #6)
#2 DIV(#1, #5)
#3 _MV_Medel <= #2
#4 OR(_MV1_L, _MV2_L)
#5 SEL(#4, 2, 1)
#6 SEL(_MV2_L, _MV2, 0)
_END_CFC_
END_FUNCTION_BLOCK

(* POU xEgna Funktionsblock/fbMONTHDAY, ST *)
FUNCTION_BLOCK fbMONTHDAY

VAR_INPUT
	_uiMonth		:UINT;
	_uiDay			:UINT;
END_VAR

VAR_OUTPUT
	uiMonthDay		:UINT;
END_VAR
uiMonthDay:=(_uiMonth*100)+_uiDay;
END_FUNCTION_BLOCK

(* POU xEgna Funktionsblock/fbOffDelayResetSO, CFC *)
FUNCTION_BLOCK fbOffDelayResetSO
VAR_INPUT
	bSO:BOOL;
	bTimerIndikering:BOOL;
	iFFD_Minuter:INT;
END_VAR
VAR_OUTPUT
	bEnable: BOOL;
END_VAR
VAR
	fbTOF1: TOF;
	fbTRIG: R_TRIG;

	HAND: BOOL:=FALSE;
	Tid: TIME;
END_VAR
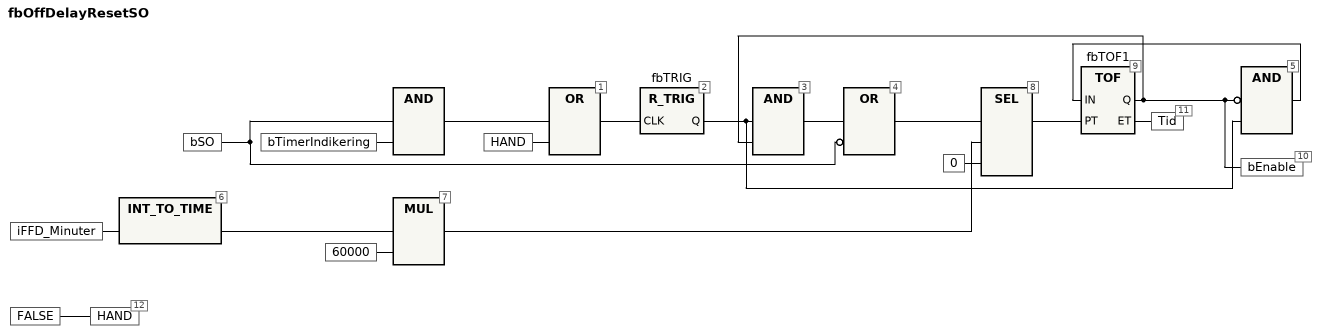
_CFC_ (* Continuous Function Chart, elements in execution order *)
#0 AND(bSO, bTimerIndikering)
#1 OR(#0, HAND)
#2 fbTRIG:R_TRIG(CLK: #1)
#3 AND(#2.Q, #9.Q)
#4 OR(#3, NOT bSO)
#5 AND(NOT #9.Q, #2.Q)
#6 INT_TO_TIME(iFFD_Minuter)
#7 MUL(#6, 60000)
#8 SEL(#4, #7, 0)
#9 fbTOF1:TOF(IN: #5, PT: #8)
#10 bEnable <= #9.Q
#11 Tid <= #9.ET
#12 HAND <= FALSE
_END_CFC_
(* the same logic as Structured Text *)
fbTRIG(CLK := (bSO AND bTimerIndikering) OR HAND);
fbTOF1(IN := NOT fbTOF1.Q AND fbTRIG.Q, PT := SEL((fbTRIG.Q AND fbTOF1.Q) OR NOT bSO, INT_TO_TIME(iFFD_Minuter) * 60000, 0));
bEnable := fbTOF1.Q;
Tid := fbTOF1.ET;
HAND := FALSE;
END_FUNCTION_BLOCK

(* POU xEgna Funktionsblock/Modbus/Modbusfunktioner_med_Master/fbReadHoldingReg_1INT, ST *)
FUNCTION_BLOCK fbReadHoldingReg_1INT
VAR
	MB_HoldingRegs					:FB_MBReadRegs;
	MB_InputRegs					:FB_MBReadInputRegs;
	fbDelay:							TON;									(*Fördröj läsning*)

	iDx									:INT:= 0;								(*Index för sekvensen*)

(* Variables used for generic handling *)
	bReturnAfterAction				:BOOL;
	bInit								:BOOL := TRUE;
	nState								:INT;
	iGenericID							:INT;
	bHasBeenBusy					:BOOL;

(*Läsvärden*)
	iReadData							:INT;									(* Läst data *)


END_VAR
VAR_INPUT
	bEnable							:BOOL;								(*Start*)
	sIPAddr	 						:STRING(15);
	uiSlaveId							:BYTE;									(*Slavadress, 255*)

(* Skicka in en pekare till controller strukten som ska vara master för denna kommunikation *)
	pController						:POINTER TO ST_TCP_CONTROLLER;	(* Pekare till strukturen *)

	wStartAddress					:WORD; 								(*Modbusadress i slav*)
	iHoldingRegOrInputReg			:INT;									(*Om inputen har värdet "0" läser man Holding Register, vid värde "1" läses Input Regs*)
	iSkalaDecimaler					:INT;									(* MIN-värde 1*)
END_VAR

VAR_OUTPUT
	bError								:BOOL;								(*Vi har ett fel*)
	bBusy								:BOOL;								(* Arbetar*)
	rReadData							:REAL;

END_VAR
actGenericHandling();
IF bReturnAfterAction THEN
	RETURN;
END_IF

CASE iDx OF

0:(*Vänta på start*)
IF
	bEnable THEN
	pController^.bUnitIsBusy:=TRUE;
	pController^.bUnitIsDone:=FALSE;
	bHasBeenBusy:=FALSE;
	bBusy:=TRUE;
		iDx := 5;
ELSIF
	bEnable AND iHoldingRegOrInputReg=1 THEN
	pController^.bUnitIsBusy:=TRUE;
	pController^.bUnitIsDone:=FALSE;
	bBusy:=TRUE;
		iDx := 10;
ELSE
	bBusy:=FALSE;
	bError:=FALSE;
END_IF


5:(*Läs holding registers. Modbus funktion 3*)
	MB_HoldingRegs(
					sIPAddr:= sIPAddr,
					nTCPPort:=502,
					nUnitID:= uiSlaveId ,
					nQuantity:= 1,
					nMBAddr:= wStartAddress ,
					cbLength:= SIZEOF(iReadData) ,
					pDestAddr:= ADR(iReadData) ,
					bExecute:= TRUE ,
					TTimeout:= T#1s ,
					bBUSY=> ,
					bError=> ,
					nErrId=> ,
					cbRead=> );

	IF NOT MB_HoldingRegs.bBusy AND NOT MB_HoldingRegs.bError THEN
		MB_HoldingRegs(bExecute:=FALSE);
		bError := FALSE;
		bBusy:=FALSE;
(*Beräkna data till utgång*)
		rReadData:= INT_TO_REAL(iReadData)/iSkalaDecimaler;
		iDx := 888;
	ELSIF MB_HoldingRegs.bError THEN
		MB_HoldingRegs(bExecute:=FALSE);
		iDx := 999;
	END_IF


10:(*Läs holding registers. Modbus funktion 3*)
	MB_InputRegs(
					sIPAddr:= sIPAddr,
					nTCPPort:=502,
					nUnitID:= uiSlaveId ,
					nQuantity:= 1,
					nMBAddr:= wStartAddress ,
					cbLength:= SIZEOF(iReadData) ,
					pDestAddr:= ADR(iReadData) ,
					bExecute:= TRUE ,
					TTimeout:= T#1s ,
					bBUSY=> ,
					bError=> ,
					nErrId=> ,
					cbRead=> );

	IF NOT MB_InputRegs.bBusy AND NOT MB_InputRegs.bError THEN
		MB_InputRegs(bExecute:=FALSE);
		bError := FALSE;
		bBusy:=FALSE;
(*Beräkna data till utgång*)
		rReadData:= INT_TO_REAL(iReadData)/iSkalaDecimaler;
		iDx := 888;
	ELSIF MB_InputRegs.bError THEN
		MB_InputRegs(bExecute:=FALSE);
		iDx := 999;
	END_IF


888: (*DONE*)
	MB_HoldingRegs(bExecute:=FALSE);
	MB_InputRegs(bExecute:=FALSE);
	pController^.bUnitIsBusy:=FALSE;
	pController^.bUnitIsDone:=TRUE;

	bBusy:=FALSE;
	iDx := 0;


999: (* Error *)
	MB_HoldingRegs(bExecute:=FALSE);
	MB_InputRegs(bExecute:=FALSE);
	bError := TRUE;
	bBusy:=FALSE;
	iDx := 1000;


1000:	(*Fördröj*)
	fbDelay(IN:= TRUE , PT:=T#2S, Q=> , ET=> );
	IF fbDelay.Q THEN
		fbDelay(IN:=FALSE);
		iDx := 888;
	END_IF

END_CASE
END_FUNCTION_BLOCK
ACTION actGenericHandling:
(* DO NOT ALTER/REMOVE *)
bReturnAfterAction:=TRUE;
(* Exit if invalid controller pointer *)
IF pController=0 THEN
	RETURN;
END_IF

(* One time initialisation *)
IF bInit THEN
	(* "Register" this block in the controller using the incremental index *)
	pController^.iNoUnits:=pController^.iNoUnits+1;
	(* Assign the generic ID of this unit *)
	iGenericID:=pController^.iNoUnits;
	(* Init done *)
	bInit:=FALSE;
END_IF

(* Exit if controller working ID doesn't match the unit ID *)
IF pController^.iWorkingUnitId<>iGenericID THEN
	RETURN;
END_IF

(* If unit isn't enabled then signal that we're done as soon as it's our turn *)
IF NOT bEnable THEN
	pController^.bUnitIsDone:=TRUE;
	pController^.bUnitIsBusy:=FALSE;
	RETURN;
END_IF

(* The code managed to get here without returning, that means we should execute the rest of the function block as well *)
bReturnAfterAction:=FALSE;
END_ACTION

(* POU xEgna Funktionsblock/Modbus/fbReadHoldingReg_1REAL, ST *)
FUNCTION_BLOCK fbReadHoldingReg_1REAL
VAR
	MB_HoldingRegs:	FB_MBReadRegs;
	uiSlaveId:				BYTE:=16#FF;						(*Modbus slavadress*)
	iDx:					INT:= 0;							(*Index för sekvensen*)

END_VAR
VAR_INPUT
	bEnable:				BOOL;								(*Start*)
	sIPAddr:	 			STRING(15);
	wAddress:				WORD; 							(*Modbusadress i slav*)

END_VAR

VAR_OUTPUT
	bError:					BOOL;								(*Vi har ett fel*)
	bBusy:					BOOL;								(* Arbetar*)

(*Läsvärden*)
	rData:					REAL;								(* Läst data*)

END_VAR
CASE iDx OF

0:(*Vänta på start*)
IF bEnable THEN
		bBusy:=TRUE;
		iDx := 5;
ELSE
		bBusy:=FALSE;
END_IF

5:(*Läs holding registers. Modbus funktion 3*)
	MB_HoldingRegs(
					sIPAddr:= sIPAddr,
					nTCPPort:=502,
					nUnitID:= uiSlaveId ,
					nQuantity:= 2,
					nMBAddr:= wAddress ,
					cbLength:= SIZEOF(rData) ,
					pDestAddr:= ADR(RData) ,
					bExecute:= TRUE ,
					TTimeout:= T#2s ,
					bBUSY=> ,
					bError=> ,
					nErrId=> ,
					cbRead=> );

	IF NOT MB_HoldingRegs.bBusy AND NOT MB_HoldingRegs.bError THEN
		MB_HoldingRegs(bExecute:=FALSE);
		bError := FALSE;
		bBusy:=FALSE;
		iDx := 0;
	ELSIF MB_HoldingRegs.bError THEN
		MB_HoldingRegs(bExecute:=FALSE);
		iDx := 999;
	END_IF

999: (* Error *)
	bError := TRUE;
	bBusy:=FALSE;
	iDx := 0;



END_CASE
END_FUNCTION_BLOCK

(* POU xEgna Funktionsblock/Modbus/Modbusfunktioner_med_Master/fbReadHoldingReg_1WORD, ST *)
FUNCTION_BLOCK fbReadHoldingReg_1WORD
VAR
	MB_HoldingRegs					:FB_MBReadRegs;
	MB_InputRegs					:FB_MBReadInputRegs;
	fbDelay:							TON;									(*Fördröj läsning*)

	iDx									:INT:= 0;								(*Index för sekvensen*)

(* Variables used for generic handling *)
	bReturnAfterAction				:BOOL;
	bInit								:BOOL := TRUE;
	nState								:INT;
	iGenericID							:INT;

(*Läsvärden*)
	wReadData							:WORD;									(* Läst data *)


END_VAR
VAR_INPUT
	bEnable							:BOOL;								(*Start*)
	sIPAddr	 						:STRING(15);
	uiSlaveId							:BYTE;									(*Slavadress, 255*)

(* Skicka in en pekare till controller strukten som ska vara master för denna kommunikation *)
	pController						:POINTER TO ST_TCP_CONTROLLER;	(* Pekare till strukturen *)

	wStartAddress					:WORD; 								(*Modbusadress i slav*)

	iHoldingRegOrInputReg			:INT;									(*Om inputen har värdet "0" läser man Holding Register, vid värde "1" läses Input Regs*)
	iSkalaDecimaler					:INT;									(* MIN-värde 1*)
END_VAR

VAR_OUTPUT
	bError								:BOOL;								(*Vi har ett fel*)
	bBusy								:BOOL;								(* Arbetar*)
	rReadData							:REAL;
	iReadDataOut						:INT;
END_VAR
actGenericHandling();
IF bReturnAfterAction THEN
	RETURN;
END_IF

CASE iDx OF

0:(*Vänta på start*)
IF
	bEnable THEN
	pController^.bUnitIsBusy:=TRUE;
	pController^.bUnitIsDone:=FALSE;
	bBusy:=TRUE;
		iDx := 5;
ELSIF
	bEnable AND iHoldingRegOrInputReg=1 THEN
	pController^.bUnitIsBusy:=TRUE;
	pController^.bUnitIsDone:=FALSE;
	bBusy:=TRUE;
		iDx := 10;
ELSE
	bBusy:=FALSE;
	bError:=FALSE;
END_IF


5:(*Läs holding registers. Modbus funktion 3*)
	MB_HoldingRegs(
					sIPAddr:= sIPAddr,
					nTCPPort:=502,
					nUnitID:= uiSlaveId ,
					nQuantity:= 1,
					nMBAddr:= wStartAddress ,
					cbLength:= SIZEOF(wReadData) ,
					pDestAddr:= ADR(wReadData) ,
					bExecute:= TRUE ,
					TTimeout:= T#1s ,
					bBUSY=> ,
					bError=> ,
					nErrId=> ,
					cbRead=> );

	IF NOT MB_HoldingRegs.bBusy AND NOT MB_HoldingRegs.bError THEN
		MB_HoldingRegs(bExecute:=FALSE);
		bError := FALSE;
		bBusy:=FALSE;

(*Beräkna data till utgång*)
		rReadData:= WORD_TO_REAL(wReadData)/iSkalaDecimaler;
		iReadDataOut:= WORD_TO_INT(wReadData)/iSkalaDecimaler;
		iDx := 888;
	ELSIF MB_HoldingRegs.bError THEN
		MB_HoldingRegs(bExecute:=FALSE);
		iDx := 999;
	END_IF


(*	IF MB_HoldingRegs.bBusy THEN
		bHasBeenBusy:=TRUE;
	ELSE
		IF bHasBeenBusy THEN
			IF NOT MB_HoldingRegs.bError THEN
				bError:=FALSE;
				iDx := 888;
			ELSE
				iDx := 999;
			END_IF
					MB_HoldingRegs(bExecute:=FALSE);
		END_IF
	END_IF
*)

10:(*Läs holding registers. Modbus funktion 3*)
	MB_InputRegs(
					sIPAddr:= sIPAddr,
					nTCPPort:=502,
					nUnitID:= uiSlaveId ,
					nQuantity:= 1,
					nMBAddr:= wStartAddress ,
					cbLength:= SIZEOF(wReadData) ,
					pDestAddr:= ADR(wReadData) ,
					bExecute:= TRUE ,
					TTimeout:= T#1s ,
					bBUSY=> ,
					bError=> ,
					nErrId=> ,
					cbRead=> );

	IF NOT MB_InputRegs.bBusy AND NOT MB_InputRegs.bError THEN
		MB_InputRegs(bExecute:=FALSE);
		bError := FALSE;
		bBusy:=FALSE;

(*Beräkna data till utgång*)
		rReadData:= WORD_TO_REAL(wReadData)/iSkalaDecimaler;
		iReadDataOut:= WORD_TO_INT(wReadData)/iSkalaDecimaler;
		iDx := 888;
	ELSIF MB_InputRegs.bError THEN
		MB_InputRegs(bExecute:=FALSE);
		iDx := 999;
	END_IF


888: (*DONE*)
	MB_HoldingRegs(bExecute:=FALSE);
	MB_InputRegs(bExecute:=FALSE);
	pController^.bUnitIsBusy:=FALSE;
	pController^.bUnitIsDone:=TRUE;

	bBusy:=FALSE;
	iDx := 0;


999: (* Error *)
	MB_HoldingRegs(bExecute:=FALSE);
	MB_InputRegs(bExecute:=FALSE);
	bError := TRUE;
	bBusy:=FALSE;
	iDx := 1000;


1000:	(*Fördröj*)
	fbDelay(IN:= TRUE , PT:=T#500ms, Q=> , ET=> );
	IF fbDelay.Q THEN
		fbDelay(IN:=FALSE);
		iDx := 888;
	END_IF

END_CASE
END_FUNCTION_BLOCK
ACTION actGenericHandling:
(* DO NOT ALTER/REMOVE *)
bReturnAfterAction:=TRUE;
(* Exit if invalid controller pointer *)
IF pController=0 THEN
	RETURN;
END_IF

(* One time initialisation *)
IF bInit THEN
	(* "Register" this block in the controller using the incremental index *)
	pController^.iNoUnits:=pController^.iNoUnits+1;
	(* Assign the generic ID of this unit *)
	iGenericID:=pController^.iNoUnits;
	(* Init done *)
	bInit:=FALSE;
END_IF

(* Exit if controller working ID doesn't match the unit ID *)
IF pController^.iWorkingUnitId<>iGenericID THEN
	RETURN;
END_IF

(* If unit isn't enabled then signal that we're done as soon as it's our turn *)
IF NOT bEnable THEN
	pController^.bUnitIsDone:=TRUE;
	pController^.bUnitIsBusy:=FALSE;
	RETURN;
END_IF

(* The code managed to get here without returning, that means we should execute the rest of the function block as well *)
bReturnAfterAction:=FALSE;
END_ACTION

(* POU xEgna Funktionsblock/Modbus/Modbusfunktioner_med_Master/fbReadHoldingReg_INT, ST *)
FUNCTION_BLOCK fbReadHoldingReg_INT
VAR
	MB_HoldingRegs					:FB_MBReadRegs;
	MB_InputRegs					:FB_MBReadInputRegs;
	fbDelay:							TON;									(*Fördröj läsning*)

	iDx									:INT:= 0;								(*Index för sekvensen*)

(* Variables used for generic handling *)
	bReturnAfterAction				:BOOL;
	bInit								:BOOL := TRUE;
	nState								:INT;
	iGenericID							:INT;

(*Läsvärden*)
	iReadDataArray					:ARRAY[0..19]		OF	INT;			(* Läst data, MAX 20 register *)


END_VAR
VAR_INPUT
	bEnable							:BOOL;								(*Start*)
	sIPAddr	 						:STRING(15);
	uiSlaveId							:BYTE;									(*Slavadress, 255*)

(* Skicka in en pekare till controller strukten som ska vara master för denna kommunikation *)
	pController						:POINTER TO ST_TCP_CONTROLLER;	(* Pekare till strukturen *)

	wStartAddress					:WORD; 								(*Modbusadress i slav*)
	wQuantity							:WORD;
	iHoldingRegOrInputReg			:INT;									(*Om inputen har värdet "0" läser man Holding Register, vid värde "1" läses Input Regs*)

END_VAR

VAR_OUTPUT
	bError								:BOOL;								(*Vi har ett fel*)
	bBusy								:BOOL;								(* Arbetar*)

END_VAR
actGenericHandling();
IF bReturnAfterAction THEN
	RETURN;
END_IF

CASE iDx OF

0:(*Vänta på start*)
IF
	bEnable THEN
	pController^.bUnitIsBusy:=TRUE;
	pController^.bUnitIsDone:=FALSE;
	bBusy:=TRUE;
		iDx := 5;
ELSIF
	bEnable AND iHoldingRegOrInputReg=1 THEN
	pController^.bUnitIsBusy:=TRUE;
	pController^.bUnitIsDone:=FALSE;
	bBusy:=TRUE;
		iDx := 10;
ELSE
	bBusy:=FALSE;
	bError:=FALSE;
END_IF


5:(*Läs holding registers. Modbus funktion 3*)
	MB_HoldingRegs(
					sIPAddr:= sIPAddr,
					nTCPPort:=502,
					nUnitID:= uiSlaveId ,
					nQuantity:= wQuantity,
					nMBAddr:= wStartAddress ,
					cbLength:= SIZEOF(iReadDataArray) ,
					pDestAddr:= ADR(iReadDataArray) ,
					bExecute:= TRUE ,
					TTimeout:= T#1s ,
					bBUSY=> ,
					bError=> ,
					nErrId=> ,
					cbRead=> );

	IF NOT MB_HoldingRegs.bBusy AND NOT MB_HoldingRegs.bError THEN
		MB_HoldingRegs(bExecute:=FALSE);
		bError := FALSE;
		bBusy:=FALSE;
		iDx := 888;
	ELSIF MB_HoldingRegs.bError THEN
		MB_HoldingRegs(bExecute:=FALSE);
		iDx := 999;
	END_IF


10:(*Läs holding registers. Modbus funktion 3*)
	MB_InputRegs(
					sIPAddr:= sIPAddr,
					nTCPPort:=502,
					nUnitID:= uiSlaveId ,
					nQuantity:= wQuantity,
					nMBAddr:= wStartAddress ,
					cbLength:= SIZEOF(iReadDataArray) ,
					pDestAddr:= ADR(iReadDataArray) ,
					bExecute:= TRUE ,
					TTimeout:= T#1s ,
					bBUSY=> ,
					bError=> ,
					nErrId=> ,
					cbRead=> );

	IF NOT MB_InputRegs.bBusy AND NOT MB_InputRegs.bError THEN
		MB_InputRegs(bExecute:=FALSE);
		bError := FALSE;
		bBusy:=FALSE;
		iDx := 888;
	ELSIF MB_InputRegs.bError THEN
		MB_InputRegs(bExecute:=FALSE);
		iDx := 999;
	END_IF


888: (*DONE*)
	MB_HoldingRegs(bExecute:=FALSE);
	MB_InputRegs(bExecute:=FALSE);
	pController^.bUnitIsBusy:=FALSE;
	pController^.bUnitIsDone:=TRUE;

	bBusy:=FALSE;
	iDx := 0;


999: (* Error *)
	MB_HoldingRegs(bExecute:=FALSE);
	MB_InputRegs(bExecute:=FALSE);
	bError := TRUE;
	bBusy:=FALSE;
	iDx := 1000;


1000:	(*Fördröj*)
	fbDelay(IN:= TRUE , PT:=T#500MS, Q=> , ET=> );
	IF fbDelay.Q THEN
		fbDelay(IN:=FALSE);
		iDx := 888;
	END_IF



END_CASE
END_FUNCTION_BLOCK
ACTION actGenericHandling:
(* DO NOT ALTER/REMOVE *)
bReturnAfterAction:=TRUE;
(* Exit if invalid controller pointer *)
IF pController=0 THEN
	RETURN;
END_IF

(* One time initialisation *)
IF bInit THEN
	(* "Register" this block in the controller using the incremental index *)
	pController^.iNoUnits:=pController^.iNoUnits+1;
	(* Assign the generic ID of this unit *)
	iGenericID:=pController^.iNoUnits;
	(* Init done *)
	bInit:=FALSE;
END_IF

(* Exit if controller working ID doesn't match the unit ID *)
IF pController^.iWorkingUnitId<>iGenericID THEN
	RETURN;
END_IF

(* If unit isn't enabled then signal that we're done as soon as it's our turn *)
IF NOT bEnable THEN
	pController^.bUnitIsDone:=TRUE;
	pController^.bUnitIsBusy:=FALSE;
	RETURN;
END_IF

(* The code managed to get here without returning, that means we should execute the rest of the function block as well *)
bReturnAfterAction:=FALSE;
END_ACTION

(* POU xEgna Funktionsblock/Modbus/Modbusfunktioner_med_Master/fbReadHoldingReg_REAL, ST *)
FUNCTION_BLOCK fbReadHoldingReg_REAL
VAR
	MB_HoldingRegs					:FB_MBReadRegs;
	MB_InputRegs					:FB_MBReadInputRegs;
	fbDelay:							TON;									(*Fördröj läsning*)

	iDx									:INT:= 0;								(*Index för sekvensen*)
	CalcQuantity						:WORD;

(* Variables used for generic handling *)
	bReturnAfterAction				:BOOL;
	bInit								:BOOL := TRUE;
	nState								:INT;
	iGenericID							:INT;

(*Läsvärden*)
	rReadDataArray					:ARRAY[0..19]		OF	REAL;			(* Läst data, MAX 20 register *)


END_VAR
VAR_INPUT
	bEnable							:BOOL;								(*Start*)
	sIPAddr	 						:STRING(15);
	uiSlaveId							:BYTE;									(*Slavadress, 255*)

(* Skicka in en pekare till controller strukten som ska vara master för denna kommunikation *)
	pController						:POINTER TO ST_TCP_CONTROLLER;	(* Pekare till strukturen *)

	wStartAddress					:WORD; 								(*Modbusadress i slav*)
	wQuantity							:WORD;
	iHoldingRegOrInputReg			:INT;									(*Om inputen har värdet "0" läser man Holding Register, vid värde "1" läses Input Regs*)

END_VAR

VAR_OUTPUT
	bError								:BOOL;								(*Vi har ett fel*)
	bBusy								:BOOL;								(* Arbetar*)

END_VAR
CalcQuantity:= wQuantity*2;

actGenericHandling();
IF bReturnAfterAction THEN
	RETURN;
END_IF

CASE iDx OF

0:(*Vänta på start*)
IF
	bEnable THEN
	pController^.bUnitIsBusy:=TRUE;
	pController^.bUnitIsDone:=FALSE;
	bBusy:=TRUE;
		iDx := 5;
ELSIF
	bEnable AND iHoldingRegOrInputReg=1 THEN
	pController^.bUnitIsBusy:=TRUE;
	pController^.bUnitIsDone:=FALSE;
	bBusy:=TRUE;
		iDx := 10;
ELSE
	bBusy:=FALSE;
	bError:=FALSE;
END_IF


5:(*Läs holding registers. Modbus funktion 3*)
	MB_HoldingRegs(
					sIPAddr:= sIPAddr,
					nTCPPort:=502,
					nUnitID:= uiSlaveId ,
					nQuantity:= CalcQuantity,
					nMBAddr:= wStartAddress ,
					cbLength:= SIZEOF(rReadDataArray) ,
					pDestAddr:= ADR(rReadDataArray) ,
					bExecute:= TRUE ,
					TTimeout:= T#1s ,
					bBUSY=> ,
					bError=> ,
					nErrId=> ,
					cbRead=> );

	IF NOT MB_HoldingRegs.bBusy AND NOT MB_HoldingRegs.bError THEN
		MB_HoldingRegs(bExecute:=FALSE);
		bError := FALSE;
		bBusy:=FALSE;
		iDx := 888;
	ELSIF MB_HoldingRegs.bError THEN
		MB_HoldingRegs(bExecute:=FALSE);
		iDx := 999;
	END_IF


10:(*Läs holding registers. Modbus funktion 3*)
	MB_InputRegs(
					sIPAddr:= sIPAddr,
					nTCPPort:=502,
					nUnitID:= uiSlaveId ,
					nQuantity:= wQuantity,
					nMBAddr:= wStartAddress ,
					cbLength:= SIZEOF(rReadDataArray) ,
					pDestAddr:= ADR(rReadDataArray) ,
					bExecute:= TRUE ,
					TTimeout:= T#1s ,
					bBUSY=> ,
					bError=> ,
					nErrId=> ,
					cbRead=> );

	IF NOT MB_InputRegs.bBusy AND NOT MB_InputRegs.bError THEN
		MB_InputRegs(bExecute:=FALSE);
		bError := FALSE;
		bBusy:=FALSE;
		iDx := 888;
	ELSIF MB_InputRegs.bError THEN
		MB_InputRegs(bExecute:=FALSE);
		iDx := 999;
	END_IF


888: (*DONE*)
	MB_HoldingRegs(bExecute:=FALSE);
	MB_InputRegs(bExecute:=FALSE);
	pController^.bUnitIsBusy:=FALSE;
	pController^.bUnitIsDone:=TRUE;
	MB_HoldingRegs(bExecute:=FALSE);
	MB_InputRegs(bExecute:=FALSE);
	bBusy:=FALSE;
	iDx := 0;


999: (* Error *)

	bError := TRUE;
	bBusy:=FALSE;
	iDx := 1000;


1000:	(*Fördröj*)
	fbDelay(IN:= TRUE , PT:=T#500MS, Q=> , ET=> );
	IF fbDelay.Q THEN
		fbDelay(IN:=FALSE);
		iDx := 888;
	END_IF



END_CASE
END_FUNCTION_BLOCK
ACTION actGenericHandling:
(* DO NOT ALTER/REMOVE *)
bReturnAfterAction:=TRUE;
(* Exit if invalid controller pointer *)
IF pController=0 THEN
	RETURN;
END_IF

(* One time initialisation *)
IF bInit THEN
	(* "Register" this block in the controller using the incremental index *)
	pController^.iNoUnits:=pController^.iNoUnits+1;
	(* Assign the generic ID of this unit *)
	iGenericID:=pController^.iNoUnits;
	(* Init done *)
	bInit:=FALSE;
END_IF

(* Exit if controller working ID doesn't match the unit ID *)
IF pController^.iWorkingUnitId<>iGenericID THEN
	RETURN;
END_IF

(* If unit isn't enabled then signal that we're done as soon as it's our turn *)
IF NOT bEnable THEN
	pController^.bUnitIsDone:=TRUE;
	pController^.bUnitIsBusy:=FALSE;
	RETURN;
END_IF

(* The code managed to get here without returning, that means we should execute the rest of the function block as well *)
bReturnAfterAction:=FALSE;
END_ACTION

(* POU xEgna Funktionsblock/Modbus/Modbusfunktioner_med_Master/fbReadHoldingReg_WORD, ST *)
FUNCTION_BLOCK fbReadHoldingReg_WORD
VAR
	MB_HoldingRegs					:FB_MBReadRegs;
	MB_InputRegs					:FB_MBReadInputRegs;
	fbDelay:							TON;									(*Fördröj läsning*)

	iDx									:INT:= 0;								(*Index för sekvensen*)

(* Variables used for generic handling *)
	bReturnAfterAction				:BOOL;
	bInit								:BOOL := TRUE;
	nState								:INT;
	iGenericID							:INT;

(*Läsvärden*)
	wReadDataArray					:ARRAY[0..19]		OF	WORD;			(* Läst data, MAX 20 register *)


END_VAR
VAR_INPUT
	bEnable							:BOOL;								(*Start*)
	sIPAddr	 						:STRING(15);
	uiSlaveId							:BYTE;									(*Slavadress, 255*)

(* Skicka in en pekare till controller strukten som ska vara master för denna kommunikation *)
	pController						:POINTER TO ST_TCP_CONTROLLER;	(* Pekare till strukturen *)

	wStartAddress					:WORD; 								(*Modbusadress i slav*)
	wQuantity							:WORD;
	iHoldingRegOrInputReg			:INT;									(*Om inputen har värdet "0" läser man Holding Register, vid värde "1" läses Input Regs*)

END_VAR

VAR_OUTPUT
	bError								:BOOL;								(*Vi har ett fel*)
	bBusy								:BOOL;								(* Arbetar*)

END_VAR
actGenericHandling();
IF bReturnAfterAction THEN
	RETURN;
END_IF

CASE iDx OF

0:(*Vänta på start*)
IF
	bEnable THEN
	pController^.bUnitIsBusy:=TRUE;
	pController^.bUnitIsDone:=FALSE;
	bBusy:=TRUE;
		iDx := 5;
ELSIF
	bEnable AND iHoldingRegOrInputReg=1 THEN
	pController^.bUnitIsBusy:=TRUE;
	pController^.bUnitIsDone:=FALSE;
	bBusy:=TRUE;
		iDx := 10;
ELSE
	bBusy:=FALSE;
	bError:=FALSE;
END_IF


5:(*Läs holding registers. Modbus funktion 3*)
	MB_HoldingRegs(
					sIPAddr:= sIPAddr,
					nTCPPort:=502,
					nUnitID:= uiSlaveId ,
					nQuantity:= wQuantity,
					nMBAddr:= wStartAddress ,
					cbLength:= SIZEOF(wReadDataArray) ,
					pDestAddr:= ADR(wReadDataArray) ,
					bExecute:= TRUE ,
					TTimeout:= T#1s ,
					bBUSY=> ,
					bError=> ,
					nErrId=> ,
					cbRead=> );

	IF NOT MB_HoldingRegs.bBusy AND NOT MB_HoldingRegs.bError THEN
		MB_HoldingRegs(bExecute:=FALSE);
		bError := FALSE;
		bBusy:=FALSE;
		iDx := 888;
	ELSIF MB_HoldingRegs.bError THEN
		MB_HoldingRegs(bExecute:=FALSE);
		iDx := 999;
	END_IF


10:(*Läs holding registers. Modbus funktion 3*)
	MB_InputRegs(
					sIPAddr:= sIPAddr,
					nTCPPort:=502,
					nUnitID:= uiSlaveId ,
					nQuantity:= wQuantity,
					nMBAddr:= wStartAddress ,
					cbLength:= SIZEOF(wReadDataArray) ,
					pDestAddr:= ADR(wReadDataArray) ,
					bExecute:= TRUE ,
					TTimeout:= T#1s ,
					bBUSY=> ,
					bError=> ,
					nErrId=> ,
					cbRead=> );

	IF NOT MB_InputRegs.bBusy AND NOT MB_InputRegs.bError THEN
		MB_InputRegs(bExecute:=FALSE);
		bError := FALSE;
		bBusy:=FALSE;
		iDx := 888;
	ELSIF MB_InputRegs.bError THEN
		MB_InputRegs(bExecute:=FALSE);
		iDx := 999;
	END_IF


888: (*DONE*)
	MB_HoldingRegs(bExecute:=FALSE);
	MB_InputRegs(bExecute:=FALSE);
	pController^.bUnitIsBusy:=FALSE;
	pController^.bUnitIsDone:=TRUE;

	bBusy:=FALSE;
	iDx := 0;


999: (* Error *)
	MB_HoldingRegs(bExecute:=FALSE);
	MB_InputRegs(bExecute:=FALSE);
	bError := TRUE;
	bBusy:=FALSE;
	iDx := 1000;


1000:	(*Fördröj*)
	fbDelay(IN:= TRUE , PT:=T#500MS, Q=> , ET=> );
	IF fbDelay.Q THEN
		fbDelay(IN:=FALSE);
		iDx := 888;
	END_IF



END_CASE
END_FUNCTION_BLOCK
ACTION actGenericHandling:
(* DO NOT ALTER/REMOVE *)
bReturnAfterAction:=TRUE;
(* Exit if invalid controller pointer *)
IF pController=0 THEN
	RETURN;
END_IF

(* One time initialisation *)
IF bInit THEN
	(* "Register" this block in the controller using the incremental index *)
	pController^.iNoUnits:=pController^.iNoUnits+1;
	(* Assign the generic ID of this unit *)
	iGenericID:=pController^.iNoUnits;
	(* Init done *)
	bInit:=FALSE;
END_IF

(* Exit if controller working ID doesn't match the unit ID *)
IF pController^.iWorkingUnitId<>iGenericID THEN
	RETURN;
END_IF

(* If unit isn't enabled then signal that we're done as soon as it's our turn *)
IF NOT bEnable THEN
	pController^.bUnitIsDone:=TRUE;
	pController^.bUnitIsBusy:=FALSE;
	RETURN;
END_IF

(* The code managed to get here without returning, that means we should execute the rest of the function block as well *)
bReturnAfterAction:=FALSE;
END_ACTION

(* POU xEgna Funktionsblock/Modbus/Modbusfunktioner_med_Master/fbWriteHoldingReg_INT, ST *)
FUNCTION_BLOCK fbWriteHoldingReg_INT
VAR
	MB_HoldingRegs					:FB_MBReadRegs;
	MB_WriteHoldinReg				:FB_MBWriteSingleReg;
	fbDelay:							TON;									(*Fördröj läsning*)

	iDx									:INT:= 0;								(*Index för sekvensen*)
	iDx_Next							:INT:=0;

(* Variables used for generic handling *)
	bReturnAfterAction				:BOOL;
	bInit								:BOOL := TRUE;
	nState								:INT;
	iGenericID							:INT;

(*Skrivvariabler*)
	wWriteMbAdrReg					:WORD;   							(* Adress att skriva till *)
	wWriteDataReg					:INT;							(* Data att skriva till slaven *)

(*Läsvärde*)
	iReadWriteData					:INT;								(*Läst data*)

(*Minnesvariabel*)
	rData_temp						:REAL;

END_VAR
VAR_INPUT
	bEnable							:BOOL;								(*Aktiverae läs*)
	bEnableWrite						:BOOL;								(*Aktivera skrivfunktion*)
	sIPAddr	 						:STRING(15);
	uiSlaveId							:BYTE;									(*Slavadress, 255*)

(* Skicka in en pekare till controller strukten som ska vara master för denna kommunikation *)
	pController						:POINTER TO ST_TCP_CONTROLLER;	(* Pekare till strukturen *)

	wStartAddress					:WORD; 								(*Modbusadress i slav*)
	iSkalaDecimaler					:INT;									(* MIN-värde 1*)

END_VAR

VAR_IN_OUT
	rData								:REAL;

END_VAR

VAR_OUTPUT
	bError								:BOOL;								(*Vi har ett fel*)
	bBusy								:BOOL;								(* Arbetar*)

END_VAR
actGenericHandling();
IF bReturnAfterAction THEN
	RETURN;
END_IF

CASE iDx OF

0:(*Vänta på start*)
IF
	bEnable THEN
	pController^.bUnitIsBusy:=TRUE;
	pController^.bUnitIsDone:=FALSE;
	bBusy:=TRUE;
		iDx := 5;
ELSE
	bBusy:=FALSE;
	bError:=FALSE;
END_IF


5: (*Läs holding registers. Modbus funktion 3*)
	MB_HoldingRegs(
					sIPAddr:= sIPAddr,
					nTCPPort:=502,
					nUnitID:= uiSlaveId ,
					nQuantity:= 1,
					nMBAddr:= wStartAddress ,
					cbLength:= SIZEOF(iReadWriteData) ,
					pDestAddr:= ADR(iReadWriteData) ,
					bExecute:= TRUE ,
					TTimeout:= T#1s ,
					bBUSY=> ,
					bError=> ,
					nErrId=> ,
					cbRead=> );

	IF NOT MB_HoldingRegs.bBusy AND NOT MB_HoldingRegs.bError THEN
		MB_HoldingRegs(bExecute:=FALSE);
		bError := FALSE;
		bBusy:=FALSE;
		iDx := 10;
	ELSIF MB_HoldingRegs.bError THEN
		MB_HoldingRegs(bExecute:=FALSE);
		iDx := 999;
	END_IF



10: (*Anropa actions och kontrollera om skrivning behövs*)
	fbWriteHoldingReg_INT.actCheckWrite;



50: (*Skriv data*)
MB_WriteHoldinReg(
				sIPAddr:= sIPAddr,
				nTCPPort:=502,
				nUnitID:= uiSlaveId ,
				nMBAddr:= wWriteMbAdrReg ,
				nValue:= wWriteDataReg ,
				bExecute:= TRUE ,
				TTimeout:= T#1s ,
				bBUSY=> ,
				bError=> ,
				nErrId=> );

	IF NOT MB_WriteHoldinReg.bBusy AND NOT MB_WriteHoldinReg.bError THEN
		MB_WriteHoldinReg(bExecute:=FALSE);
		bError := FALSE;
		bBusy:=FALSE;
		iDx := iDx_Next;

	ELSIF MB_WriteHoldinReg.bError THEN
		MB_WriteHoldinReg(bExecute:=FALSE);
		iDx := 999;
	END_IF


888: (*DONE*)
	MB_HoldingRegs(bExecute:=FALSE);
	MB_WriteHoldinReg(bExecute:=FALSE);
	pController^.bUnitIsBusy:=FALSE;
	pController^.bUnitIsDone:=TRUE;

	bBusy:=FALSE;
	iDx := 0;


999: (* Error *)
	MB_HoldingRegs(bExecute:=FALSE);
	MB_WriteHoldinReg(bExecute:=FALSE);
	bError := TRUE;
	bBusy:=FALSE;
	iDx := 1000;


1000:	(*Fördröj*)
	fbDelay(IN:= TRUE , PT:=T#2S, Q=> , ET=> );
	IF fbDelay.Q THEN
		fbDelay(IN:=FALSE);
		iDx := 888;
	END_IF



END_CASE
END_FUNCTION_BLOCK
ACTION actCheckWrite:
IF
	bEnableWrite AND
	rData_temp<>rData
THEN
	rData_temp:=rData;

	wWriteMbAdrReg := wStartAddress;
	wWriteDataReg := REAL_TO_INT(rData_temp*iSkalaDecimaler);
	iDx_Next:= 888;
	iDx := 50;

ELSIF

	iReadWriteData<>REAL_TO_INT(rData_temp*iSkalaDecimaler) 

THEN
	rData_temp:=INT_TO_REAL(iReadWriteData)/iSkalaDecimaler;
	rData:=INT_TO_REAL(iReadWriteData)/iSkalaDecimaler;
	iDx:=888;

ELSE
	iDx := 888;
END_IF
END_ACTION
ACTION actGenericHandling:
(* DO NOT ALTER/REMOVE *)
bReturnAfterAction:=TRUE;
(* Exit if invalid controller pointer *)
IF pController=0 THEN
	RETURN;
END_IF

(* One time initialisation *)
IF bInit THEN
	(* "Register" this block in the controller using the incremental index *)
	pController^.iNoUnits:=pController^.iNoUnits+1;
	(* Assign the generic ID of this unit *)
	iGenericID:=pController^.iNoUnits;
	(* Init done *)
	bInit:=FALSE;
END_IF

(* Exit if controller working ID doesn't match the unit ID *)
IF pController^.iWorkingUnitId<>iGenericID THEN
	RETURN;
END_IF

(* If unit isn't enabled then signal that we're done as soon as it's our turn *)
IF NOT bEnable THEN
	pController^.bUnitIsDone:=TRUE;
	pController^.bUnitIsBusy:=FALSE;
	RETURN;
END_IF

(* The code managed to get here without returning, that means we should execute the rest of the function block as well *)
bReturnAfterAction:=FALSE;
END_ACTION

(* POU xEgna Funktionsblock/Modbus/Modbusfunktioner_med_Master/fbWriteHoldingReg_INT2, ST *)
FUNCTION_BLOCK fbWriteHoldingReg_INT2
VAR
	MB_HoldingRegs					:FB_MBReadRegs;
	MB_WriteHoldinReg				:FB_MBWriteSingleReg;
	fbDelay:							TON;									(*Fördröj läsning*)

	iDx									:INT:= 0;								(*Index för sekvensen*)
	iDx_Next							:INT:=0;

(* Variables used for generic handling *)
	bReturnAfterAction				:BOOL;
	bInit								:BOOL := TRUE;
	nState								:INT;
	iGenericID							:INT;

(*Skrivvariabler*)
	wWriteMbAdrReg					:WORD;   							(* Adress att skriva till *)
	wWriteDataReg					:INT;							(* Data att skriva till slaven *)

(*Läsvärde*)
	iReadWriteData					:INT;								(*Läst data*)

(*Minnesvariabel*)
	iData_temp						:INT;

END_VAR
VAR_INPUT
	bEnable							:BOOL;								(*Aktiverae läs*)
	bEnableWrite						:BOOL;								(*Aktivera skrivfunktion*)
	sIPAddr	 						:STRING(15);
	uiSlaveId							:BYTE;									(*Slavadress, 255*)

(* Skicka in en pekare till controller strukten som ska vara master för denna kommunikation *)
	pController						:POINTER TO ST_TCP_CONTROLLER;	(* Pekare till strukturen *)

	wStartAddress					:WORD; 								(*Modbusadress i slav*)
	iSkalaDecimaler					:INT;									(* MIN-värde 1*)

END_VAR

VAR_IN_OUT
	iData								:INT;

END_VAR

VAR_OUTPUT
	bError								:BOOL;								(*Vi har ett fel*)
	bBusy								:BOOL;								(* Arbetar*)

END_VAR
actGenericHandling();
IF bReturnAfterAction THEN
	RETURN;
END_IF

CASE iDx OF

0:(*Vänta på start*)
IF
	bEnable THEN
	pController^.bUnitIsBusy:=TRUE;
	pController^.bUnitIsDone:=FALSE;
	bBusy:=TRUE;
		iDx := 5;
ELSE
	bBusy:=FALSE;
	bError:=FALSE;
END_IF


5: (*Läs holding registers. Modbus funktion 3*)
	MB_HoldingRegs(
					sIPAddr:= sIPAddr,
					nTCPPort:=502,
					nUnitID:= uiSlaveId ,
					nQuantity:= 1,
					nMBAddr:= wStartAddress ,
					cbLength:= SIZEOF(iReadWriteData) ,
					pDestAddr:= ADR(iReadWriteData) ,
					bExecute:= TRUE ,
					TTimeout:= T#1s ,
					bBUSY=> ,
					bError=> ,
					nErrId=> ,
					cbRead=> );

	IF NOT MB_HoldingRegs.bBusy AND NOT MB_HoldingRegs.bError THEN
		MB_HoldingRegs(bExecute:=FALSE);
		bError := FALSE;
		bBusy:=FALSE;
		iDx := 10;
	ELSIF MB_HoldingRegs.bError THEN
		MB_HoldingRegs(bExecute:=FALSE);
		iDx := 999;
	END_IF



10: (*Anropa actions och kontrollera om skrivning behövs*)
	fbWriteHoldingReg_INT2.actCheckWrite;



50: (*Skriv data*)
MB_WriteHoldinReg(
				sIPAddr:= sIPAddr,
				nTCPPort:=502,
				nUnitID:= uiSlaveId ,
				nMBAddr:= wWriteMbAdrReg ,
				nValue:= wWriteDataReg ,
				bExecute:= TRUE ,
				TTimeout:= T#1s ,
				bBUSY=> ,
				bError=> ,
				nErrId=> );

	IF NOT MB_WriteHoldinReg.bBusy AND NOT MB_WriteHoldinReg.bError THEN
		MB_WriteHoldinReg(bExecute:=FALSE);
		bError := FALSE;
		bBusy:=FALSE;
		iDx := iDx_Next;

	ELSIF MB_WriteHoldinReg.bError THEN
		MB_WriteHoldinReg(bExecute:=FALSE);
		iDx := 999;
	END_IF


888: (*DONE*)
	MB_HoldingRegs(bExecute:=FALSE);
	MB_WriteHoldinReg(bExecute:=FALSE);
	pController^.bUnitIsBusy:=FALSE;
	pController^.bUnitIsDone:=TRUE;

	bBusy:=FALSE;
	iDx := 0;


999: (* Error *)
	MB_HoldingRegs(bExecute:=FALSE);
	MB_WriteHoldinReg(bExecute:=FALSE);
	bError := TRUE;
	bBusy:=FALSE;
	iDx := 1000;


1000:	(*Fördröj*)
	fbDelay(IN:= TRUE , PT:=T#2s, Q=> , ET=> );
	IF fbDelay.Q THEN
		fbDelay(IN:=FALSE);
		iDx := 888;
	END_IF



END_CASE
END_FUNCTION_BLOCK
ACTION actCheckWrite:
IF
	bEnableWrite AND
	iData_temp<>iData
THEN
	iData_temp:=iData;

	wWriteMbAdrReg := wStartAddress;
	wWriteDataReg := (iData_temp*iSkalaDecimaler);
	iDx_Next:= 888;
	iDx := 50;

ELSIF

	iReadWriteData<>(iData_temp*iSkalaDecimaler)

THEN
	iData_temp:=(iReadWriteData/iSkalaDecimaler);
	iData:=(iReadWriteData/iSkalaDecimaler);
	iDx:=888;

ELSE
	iDx := 888;
END_IF
END_ACTION
ACTION actGenericHandling:
(* DO NOT ALTER/REMOVE *)
bReturnAfterAction:=TRUE;
(* Exit if invalid controller pointer *)
IF pController=0 THEN
	RETURN;
END_IF

(* One time initialisation *)
IF bInit THEN
	(* "Register" this block in the controller using the incremental index *)
	pController^.iNoUnits:=pController^.iNoUnits+1;
	(* Assign the generic ID of this unit *)
	iGenericID:=pController^.iNoUnits;
	(* Init done *)
	bInit:=FALSE;
END_IF

(* Exit if controller working ID doesn't match the unit ID *)
IF pController^.iWorkingUnitId<>iGenericID THEN
	RETURN;
END_IF

(* If unit isn't enabled then signal that we're done as soon as it's our turn *)
IF NOT bEnable THEN
	pController^.bUnitIsDone:=TRUE;
	pController^.bUnitIsBusy:=FALSE;
	RETURN;
END_IF

(* The code managed to get here without returning, that means we should execute the rest of the function block as well *)
bReturnAfterAction:=FALSE;
END_ACTION

(* POU xEgna Funktionsblock/Modbus/Modbusfunktioner_med_Master/fbWriteHoldingReg_WORD, ST *)
FUNCTION_BLOCK fbWriteHoldingReg_WORD
VAR
	MB_HoldingRegs					:FB_MBReadRegs;
	MB_WriteHoldinReg				:FB_MBWriteSingleReg;
	fbDelay:							TON;									(*Fördröj läsning*)

	iDx									:INT:= 0;								(*Index för sekvensen*)
	iDx_Next							:INT:=0;

(* Variables used for generic handling *)
	bReturnAfterAction				:BOOL;
	bInit								:BOOL := TRUE;
	nState								:INT;
	iGenericID							:INT;

(*Skrivvariabler*)
	wWriteMbAdrReg					:WORD;   							(* Adress att skriva till *)
	wWriteDataReg					:WORD;							(* Data att skriva till slaven *)

(*Läsvärde*)
	wReadWriteData					:WORD;								(*Läst data*)

(*Minnesvariabel*)
	rData_temp						:REAL;

END_VAR
VAR_INPUT
	bEnable							:BOOL;								(*Aktiverae läs*)
	bEnableWrite						:BOOL;								(*Aktivera skrivfunktion*)
	sIPAddr	 						:STRING(15);
	uiSlaveId							:BYTE;									(*Slavadress, 255*)

(* Skicka in en pekare till controller strukten som ska vara master för denna kommunikation *)
	pController						:POINTER TO ST_TCP_CONTROLLER;	(* Pekare till strukturen *)

	wStartAddress					:WORD; 								(*Modbusadress i slav*)
	iSkalaDecimaler					:INT;									(* MIN-värde 1*)

END_VAR

VAR_IN_OUT
	rData								:REAL;

END_VAR

VAR_OUTPUT
	bError								:BOOL;								(*Vi har ett fel*)
	bBusy								:BOOL;								(* Arbetar*)

END_VAR
actGenericHandling();
IF bReturnAfterAction THEN
	RETURN;
END_IF

CASE iDx OF

0:(*Vänta på start*)
IF
	bEnable THEN
	pController^.bUnitIsBusy:=TRUE;
	pController^.bUnitIsDone:=FALSE;
	bBusy:=TRUE;
		iDx := 5;
ELSE
	bBusy:=FALSE;
	bError:=FALSE;
END_IF


5: (*Läs holding registers. Modbus funktion 3*)
	MB_HoldingRegs(
					sIPAddr:= sIPAddr,
					nTCPPort:=502,
					nUnitID:= uiSlaveId ,
					nQuantity:= 1,
					nMBAddr:= wStartAddress ,
					cbLength:= SIZEOF(wReadWriteData) ,
					pDestAddr:= ADR(wReadWriteData) ,
					bExecute:= TRUE ,
					TTimeout:= T#1s ,
					bBUSY=> ,
					bError=> ,
					nErrId=> ,
					cbRead=> );

	IF NOT MB_HoldingRegs.bBusy AND NOT MB_HoldingRegs.bError THEN
		MB_HoldingRegs(bExecute:=FALSE);
		bError := FALSE;
		bBusy:=FALSE;
		iDx := 10;
	ELSIF MB_HoldingRegs.bError THEN
		MB_HoldingRegs(bExecute:=FALSE);
		iDx := 999;
	END_IF



10: (*Anropa actions och kontrollera om skrivning behövs*)
	fbWriteHoldingReg_WORD.actCheckWrite;



50: (*Skriv data*)
MB_WriteHoldinReg(
				sIPAddr:= sIPAddr,
				nTCPPort:=502,
				nUnitID:= uiSlaveId ,
				nMBAddr:= wWriteMbAdrReg ,
				nValue:= wWriteDataReg ,			(*				nValue:= SIZEOF(wWriteDataReg) ,*)
				bExecute:= TRUE ,
				TTimeout:= T#1s ,
				bBUSY=> ,
				bError=> ,
				nErrId=> );

	IF NOT MB_WriteHoldinReg.bBusy AND NOT MB_WriteHoldinReg.bError THEN
		MB_WriteHoldinReg(bExecute:=FALSE);
		bError := FALSE;
		bBusy:=FALSE;
		iDx := iDx_Next;

	ELSIF MB_WriteHoldinReg.bError THEN
		MB_WriteHoldinReg(bExecute:=FALSE);
		iDx := 999;
	END_IF


888: (*DONE*)
	MB_HoldingRegs(bExecute:=FALSE);
	MB_WriteHoldinReg(bExecute:=FALSE);
	pController^.bUnitIsBusy:=FALSE;
	pController^.bUnitIsDone:=TRUE;

	bBusy:=FALSE;
	iDx := 0;


999: (* Error *)
	MB_HoldingRegs(bExecute:=FALSE);
	MB_WriteHoldinReg(bExecute:=FALSE);
	bError := TRUE;
	bBusy:=FALSE;
	iDx := 1000;


1000:	(*Fördröj*)
	fbDelay(IN:= TRUE , PT:=T#2S, Q=> , ET=> );
	IF fbDelay.Q THEN
		fbDelay(IN:=FALSE);
		iDx := 888;
	END_IF


END_CASE
END_FUNCTION_BLOCK
ACTION actCheckWrite:
IF
	bEnableWrite AND
	rData_temp<>rData
THEN
	rData_temp:=rData;

	wWriteMbAdrReg := wStartAddress;
	wWriteDataReg := REAL_TO_WORD(rData_temp*iSkalaDecimaler);
	iDx_Next:= 888;
	iDx := 50;

ELSIF

	wReadWriteData<>REAL_TO_WORD(rData_temp*iSkalaDecimaler)

THEN
	rData_temp:=WORD_TO_REAL(wReadWriteData)/iSkalaDecimaler;
	rData:=WORD_TO_REAL(wReadWriteData)/iSkalaDecimaler;
	iDx:=888;

ELSE
	iDx := 888;
END_IF








(*
IF
	wReadWriteData<>REAL_TO_WORD(rData_temp*iSkalaDecimaler)

THEN
	rData_temp:=WORD_TO_REAL(wReadWriteData)/iSkalaDecimaler;
	rData:=WORD_TO_REAL(wReadWriteData)/iSkalaDecimaler;
	iDx:=888;

ELSIF
	bEnableWrite AND bError=FALSE AND
	rData_temp<>rData

THEN
	rData_temp:=rData;
	wWriteMbAdrReg := wStartAddress;
	wWriteDataReg := REAL_TO_WORD(rData_temp*iSkalaDecimaler);
	iDx_Next:= 888;
	iDx := 50;

ELSE
	iDx:=888;

END_IF

*)
END_ACTION
ACTION actGenericHandling:
(* DO NOT ALTER/REMOVE *)
bReturnAfterAction:=TRUE;
(* Exit if invalid controller pointer *)
IF pController=0 THEN
	RETURN;
END_IF

(* One time initialisation *)
IF bInit THEN
	(* "Register" this block in the controller using the incremental index *)
	pController^.iNoUnits:=pController^.iNoUnits+1;
	(* Assign the generic ID of this unit *)
	iGenericID:=pController^.iNoUnits;
	(* Init done *)
	bInit:=FALSE;
END_IF

(* Exit if controller working ID doesn't match the unit ID *)
IF pController^.iWorkingUnitId<>iGenericID THEN
	RETURN;
END_IF

(* If unit isn't enabled then signal that we're done as soon as it's our turn *)
IF NOT bEnable THEN
	pController^.bUnitIsDone:=TRUE;
	pController^.bUnitIsBusy:=FALSE;
	RETURN;
END_IF

(* The code managed to get here without returning, that means we should execute the rest of the function block as well *)
bReturnAfterAction:=FALSE;
END_ACTION

(* POU xEgna Funktionsblock/Modbus/Modbusfunktioner_med_Master/fbWriteHoldingReg_WORD2, ST *)
FUNCTION_BLOCK fbWriteHoldingReg_WORD2
VAR
	MB_HoldingRegs					:FB_MBReadRegs;
	MB_WriteHoldinReg				:FB_MBWriteSingleReg;
	fbDelay:							TON;									(*Fördröj läsning*)

	iDx									:INT:= 0;								(*Index för sekvensen*)
	iDx_Next							:INT:=0;

(* Variables used for generic handling *)
	bReturnAfterAction				:BOOL;
	bInit								:BOOL := TRUE;
	nState								:INT;
	iGenericID							:INT;

(*Skrivvariabler*)
	wWriteMbAdrReg					:WORD;   							(* Adress att skriva till *)
	wWriteDataReg					:WORD;							(* Data att skriva till slaven *)

(*Läsvärde*)
	wReadWriteData					:WORD;								(*Läst data*)

(*Minnesvariabel*)
	wData_temp						:WORD;

END_VAR
VAR_INPUT
	bEnable							:BOOL;								(*Aktiverae läs*)
	bEnableWrite						:BOOL;								(*Aktivera skrivfunktion*)
	sIPAddr	 						:STRING(15);
	uiSlaveId							:BYTE;									(*Slavadress, 255*)

(* Skicka in en pekare till controller strukten som ska vara master för denna kommunikation *)
	pController						:POINTER TO ST_TCP_CONTROLLER;	(* Pekare till strukturen *)

	wStartAddress					:WORD; 								(*Modbusadress i slav*)
	iSkalaDecimaler					:INT;									(* MIN-värde 1*)

END_VAR

VAR_IN_OUT
	wData								:WORD;

END_VAR

VAR_OUTPUT
	bError								:BOOL;								(*Vi har ett fel*)
	bBusy								:BOOL;								(* Arbetar*)

END_VAR
actGenericHandling();
IF bReturnAfterAction THEN
	RETURN;
END_IF

CASE iDx OF

0:(*Vänta på start*)
IF
	bEnable THEN
	pController^.bUnitIsBusy:=TRUE;
	pController^.bUnitIsDone:=FALSE;
	bBusy:=TRUE;
		iDx := 5;
ELSE
	bBusy:=FALSE;
	bError:=FALSE;
END_IF


5: (*Läs holding registers. Modbus funktion 3*)
	MB_HoldingRegs(
					sIPAddr:= sIPAddr,
					nTCPPort:=502,
					nUnitID:= uiSlaveId ,
					nQuantity:= 1,
					nMBAddr:= wStartAddress ,
					cbLength:= SIZEOF(wReadWriteData) ,
					pDestAddr:= ADR(wReadWriteData) ,
					bExecute:= TRUE ,
					TTimeout:= T#1s ,
					bBUSY=> ,
					bError=> ,
					nErrId=> ,
					cbRead=> );

	IF NOT MB_HoldingRegs.bBusy AND NOT MB_HoldingRegs.bError THEN
		MB_HoldingRegs(bExecute:=FALSE);
		bError := FALSE;
		bBusy:=FALSE;
		iDx := 10;
	ELSIF MB_HoldingRegs.bError THEN
		MB_HoldingRegs(bExecute:=FALSE);
		iDx := 999;
	END_IF



10: (*Anropa actions och kontrollera om skrivning behövs*)
	fbWriteHoldingReg_WORD2.actCheckWrite;



50: (*Skriv data*)
MB_WriteHoldinReg(
				sIPAddr:= sIPAddr,
				nTCPPort:=502,
				nUnitID:= uiSlaveId ,
				nMBAddr:= wWriteMbAdrReg ,
				nValue:= wWriteDataReg ,
				bExecute:= TRUE ,
				TTimeout:= T#1s ,
				bBUSY=> ,
				bError=> ,
				nErrId=> );

	IF NOT MB_WriteHoldinReg.bBusy AND NOT MB_WriteHoldinReg.bError THEN
		MB_WriteHoldinReg(bExecute:=FALSE);
		bError := FALSE;
		bBusy:=FALSE;
		iDx := iDx_Next;

	ELSIF MB_WriteHoldinReg.bError THEN
		MB_WriteHoldinReg(bExecute:=FALSE);
		iDx := 999;
	END_IF


888: (*DONE*)
	MB_HoldingRegs(bExecute:=FALSE);
	MB_WriteHoldinReg(bExecute:=FALSE);
	pController^.bUnitIsBusy:=FALSE;
	pController^.bUnitIsDone:=TRUE;

	bBusy:=FALSE;
	iDx := 0;


999: (* Error *)
	MB_HoldingRegs(bExecute:=FALSE);
	MB_WriteHoldinReg(bExecute:=FALSE);
	bError := TRUE;
	bBusy:=FALSE;
	iDx := 1000;


1000:	(*Fördröj*)
	fbDelay(IN:= TRUE , PT:=T#2s, Q=> , ET=> );
	IF fbDelay.Q THEN
		fbDelay(IN:=FALSE);
		iDx := 888;
	END_IF



END_CASE
END_FUNCTION_BLOCK
ACTION actCheckWrite:
IF
	bEnableWrite AND
	wData_temp<>wData
THEN
	wData_temp:=wData;

	wWriteMbAdrReg := wStartAddress;
	wWriteDataReg := (wData_temp*iSkalaDecimaler);
	iDx_Next:= 888;
	iDx := 50;

ELSIF
	wReadWriteData<>(wData_temp*iSkalaDecimaler)

THEN
	wData_temp:=(wReadWriteData/iSkalaDecimaler);
	wData:=(wReadWriteData/iSkalaDecimaler);
	iDx:=888;

ELSE
	iDx := 888;
END_IF
END_ACTION
ACTION actGenericHandling:
(* DO NOT ALTER/REMOVE *)
bReturnAfterAction:=TRUE;
(* Exit if invalid controller pointer *)
IF pController=0 THEN
	RETURN;
END_IF

(* One time initialisation *)
IF bInit THEN
	(* "Register" this block in the controller using the incremental index *)
	pController^.iNoUnits:=pController^.iNoUnits+1;
	(* Assign the generic ID of this unit *)
	iGenericID:=pController^.iNoUnits;
	(* Init done *)
	bInit:=FALSE;
END_IF

(* Exit if controller working ID doesn't match the unit ID *)
IF pController^.iWorkingUnitId<>iGenericID THEN
	RETURN;
END_IF

(* If unit isn't enabled then signal that we're done as soon as it's our turn *)
IF NOT bEnable THEN
	pController^.bUnitIsDone:=TRUE;
	pController^.bUnitIsBusy:=FALSE;
	RETURN;
END_IF

(* The code managed to get here without returning, that means we should execute the rest of the function block as well *)
bReturnAfterAction:=FALSE;
END_ACTION
